LIN {X 0,Y 242.038,Z 353.956,A -85,B 0,C 180,E1 -19224.498,E2 -19224.498} C_VEL
LIN {X 0,Y 241.957,Z 353.973,A -85,B 0,C 180,E1 -19228.478,E2 -19228.478} C_VEL
LIN {X 0,Y 241.972,Z 353.968,A -85,B 0,C 180,E1 -19232.309,E2 -19232.309} C_VEL
LIN {X 0,Y 242.029,Z 353.963,A -85,B 0,C 180,E1 -19236.013,E2 -19236.013} C_VEL
LIN {X 0,Y 242.039,Z 353.959,A -85,B 0,C 180,E1 -19239.608,E2 -19239.608} C_VEL
LIN {X 0,Y 242.166,Z 353.937,A -85,B 0,C 180,E1 -19243.279,E2 -19243.279} C_VEL
LIN {X 0,Y 242.184,Z 353.936,A -85,B 0,C 180,E1 -19248.28,E2 -19248.28} C_VEL
LIN {X 0,Y 242.374,Z 353.905,A -85,B 0,C 180,E1 -19251.664,E2 -19251.664} C_VEL
LIN {X 0,Y 242.4,Z 353.912,A -85,B 0,C 180,E1 -19253.341,E2 -19253.341} C_VEL
LIN {X 0,Y 242.624,Z 353.883,A -85,B 0,C 180,E1 -19258.341,E2 -19258.341} C_VEL
LIN {X 0,Y 242.63,Z 353.872,A -85,B 0,C 180,E1 -19261.66,E2 -19261.66} C_VEL
LIN {X 0,Y 242.401,Z 353.9,A -85,B 0,C 180,E1 -19266.66,E2 -19266.66} C_VEL
LIN {X 0,Y 242.268,Z 353.929,A -85,B 0,C 180,E1 -19270.024,E2 -19270.024} C_VEL
LIN {X 0,Y 242.11,Z 353.946,A -85,B 0,C 180,E1 -19275.145,E2 -19275.145} C_VEL
LIN {X 0,Y 242.019,Z 353.963,A -85,B 0,C 180,E1 -19278.629,E2 -19278.629} C_VEL
LIN {X 0,Y 241.975,Z 353.965,A -85,B 0,C 180,E1 -19282.184,E2 -19282.184} C_VEL
LIN {X 0,Y 241.988,Z 353.96,A -85,B 0,C 180,E1 -19285.827,E2 -19285.827} C_VEL
LIN {X 0,Y 241.965,Z 353.934,A -85,B 0,C 180,E1 -19289.59,E2 -19289.59} C_VEL
LIN {X 0,Y 241.982,Z 353.969,A -85,B 0,C 180,E1 -19293.493,E2 -19293.493} C_VEL
LIN {X 0,Y 241.981,Z 353.944,A -85,B 0,C 180,E1 -19297.584,E2 -19297.584} C_VEL
LIN {X 0,Y 241.974,Z 353.962,A -85,B 0,C 180,E1 -19298.682,E2 -19298.682} C_VEL
LIN {X 0,Y 242.898,Z 356.753,A -85,B 0,C 180,E1 -19299.067,E2 -19299.067} C_VEL
LIN {X 0,Y 245.049,Z 359.01,A -85,B 0,C 180,E1 -19299.727,E2 -19299.727} C_VEL
LIN {X 0,Y 247.606,Z 362.894,A -85,B 0,C 180,E1 -19300.538,E2 -19300.538} C_VEL
LIN {X 0,Y 248.987,Z 364.649,A -85,B 0,C 180,E1 -19300.949,E2 -19300.949} C_VEL
LIN {X 0,Y 256.882,Z 376.241,A -85,B 0,C 180,E1 -19303.223,E2 -19303.223} C_VEL
LIN {X 0,Y 264.702,Z 390.021,A -85,B 0,C 180,E1 -19305.346,E2 -19305.346} C_VEL
LIN {X 0,Y 272.156,Z 405.107,A -85,B 0,C 180,E1 -19307.261,E2 -19307.261} C_VEL
LIN {X 0,Y 274.978,Z 411.557,A -85,B 0,C 180,E1 -19307.97,E2 -19307.97} C_VEL
LIN {X 0,Y 271.334,Z 488.503,A -85,B 0,C 180,E1 -19309.947,E2 -19309.947} C_VEL
LIN {X 0,Y 270.043,Z 502.422,A -85,B 0,C 180,E1 -19310.566,E2 -19310.566} C_VEL
LIN {X 0,Y 267.985,Z 516.616,A -85,B 0,C 180,E1 -19311.475,E2 -19311.475} C_VEL
LIN {X 0,Y 265.359,Z 530.29,A -85,B 0,C 180,E1 -19312.664,E2 -19312.664} C_VEL
LIN {X 0,Y 262.577,Z 543.151,A -85,B 0,C 180,E1 -19314.162,E2 -19314.162} C_VEL
LIN {X 0,Y 259.471,Z 554.546,A -85,B 0,C 180,E1 -19315.803,E2 -19315.803} C_VEL
LIN {X 0,Y 256.414,Z 565.005,A -85,B 0,C 180,E1 -19317.692,E2 -19317.692} C_VEL
LIN {X 0,Y 253.24,Z 575.381,A -85,B 0,C 180,E1 -19320.03,E2 -19320.03} C_VEL
LIN {X 0,Y 250.217,Z 583.915,A -85,B 0,C 180,E1 -19322.39,E2 -19322.39} C_VEL
LIN {X 0,Y 247.608,Z 590.992,A -85,B 0,C 180,E1 -19324.801,E2 -19324.801} C_VEL
LIN {X 0,Y 245.473,Z 596.839,A -85,B 0,C 180,E1 -19327.262,E2 -19327.262} C_VEL
LIN {X 0,Y 243.185,Z 603.065,A -85,B 0,C 180,E1 -19330.588,E2 -19330.588} C_VEL
LIN {X 0,Y 241.694,Z 607.276,A -85,B 0,C 180,E1 -19333.656,E2 -19333.656} C_VEL
LIN {X 0,Y 240.668,Z 610.028,A -85,B 0,C 180,E1 -19336.49,E2 -19336.49} C_VEL
LIN {X 0,Y 239.974,Z 612.057,A -85,B 0,C 180,E1 -19339.879,E2 -19339.879} C_VEL
LIN {X 0,Y 239.855,Z 612.741,A -85,B 0,C 180,E1 -19343.269,E2 -19343.269} C_VEL
LIN {X 0,Y 239.803,Z 612.535,A -85,B 0,C 180,E1 -19345.18,E2 -19345.18} C_VEL
LIN {X 0,Y 239.895,Z 611.292,A -85,B 0,C 180,E1 -19348.321,E2 -19348.321} C_VEL
LIN {X 0,Y 240.147,Z 608.654,A -85,B 0,C 180,E1 -19351.677,E2 -19351.677} C_VEL
LIN {X 0,Y 240.892,Z 604.604,A -85,B 0,C 180,E1 -19355.021,E2 -19355.021} C_VEL
LIN {X 0,Y 242.269,Z 599.01,A -85,B 0,C 180,E1 -19358.34,E2 -19358.34} C_VEL
LIN {X 0,Y 243.69,Z 593.257,A -85,B 0,C 180,E1 -19360.994,E2 -19360.994} C_VEL
LIN {X 0,Y 245.286,Z 586.113,A -85,B 0,C 180,E1 -19363.673,E2 -19363.673} C_VEL
LIN {X 0,Y 247.415,Z 578.179,A -85,B 0,C 180,E1 -19366.079,E2 -19366.079} C_VEL
LIN {X 0,Y 249.976,Z 568.609,A -85,B 0,C 180,E1 -19368.439,E2 -19368.439} C_VEL
LIN {X 0,Y 252.356,Z 558.026,A -85,B 0,C 180,E1 -19370.585,E2 -19370.585} C_VEL
LIN {X 0,Y 254.879,Z 546.305,A -85,B 0,C 180,E1 -19372.494,E2 -19372.494} C_VEL
LIN {X 0,Y 257.449,Z 533.24,A -85,B 0,C 180,E1 -19374.172,E2 -19374.172} C_VEL
LIN {X 0,Y 259.472,Z 520.349,A -85,B 0,C 180,E1 -19375.467,E2 -19375.467} C_VEL
LIN {X 0,Y 261.277,Z 506.3,A -85,B 0,C 180,E1 -19376.51,E2 -19376.51} C_VEL
LIN {X 0,Y 262.486,Z 491.876,A -85,B 0,C 180,E1 -19377.266,E2 -19377.266} C_VEL
LIN {X 0,Y 263.407,Z 473.595,A -85,B 0,C 180,E1 -19377.827,E2 -19377.827} C_VEL
LIN {X 0,Y 266.21,Z 403.022,A -85,B 0,C 180,E1 -19379.659,E2 -19379.659} C_VEL
LIN {X 0,Y 259.511,Z 386.758,A -85,B 0,C 180,E1 -19381.142,E2 -19381.142} C_VEL
LIN {X 0,Y 253.103,Z 373.357,A -85,B 0,C 180,E1 -19382.587,E2 -19382.587} C_VEL
LIN {X 0,Y 246.089,Z 361.534,A -85,B 0,C 180,E1 -19384.184,E2 -19384.184} C_VEL
LIN {X 0,Y 243.888,Z 357.969,A -85,B 0,C 180,E1 -19384.706,E2 -19384.706} C_VEL
LIN {X 0,Y 242.341,Z 355.359,A -85,B 0,C 180,E1 -19385.085,E2 -19385.085} C_VEL
LIN {X 0,Y 242.002,Z 353.964,A -85,B 0,C 180,E1 -19385.222,E2 -19385.222} C_VEL
LIN {X 0,Y 241.996,Z 353.966,A -85,B 0,C 180,E1 -19388.359,E2 -19388.359} C_VEL
LIN {X 0,Y 241.903,Z 353.978,A -85,B 0,C 180,E1 -19393.42,E2 -19393.42} C_VEL
LIN {X 0,Y 241.909,Z 353.971,A -85,B 0,C 180,E1 -19398.071,E2 -19398.071} C_VEL
LIN {X 0,Y 241.968,Z 353.961,A -85,B 0,C 180,E1 -19402.413,E2 -19402.413} C_VEL
LIN {X 0,Y 241.981,Z 353.958,A -85,B 0,C 180,E1 -19406.507,E2 -19406.507} C_VEL
LIN {X 0,Y 241.973,Z 353.966,A -85,B 0,C 180,E1 -19410.615,E2 -19410.615} C_VEL
LIN {X 0,Y 241.998,Z 353.961,A -85,B 0,C 180,E1 -19414.197,E2 -19414.197} C_VEL
LIN {X 0,Y 241.989,Z 353.939,A -85,B 0,C 180,E1 -19418.337,E2 -19418.337} C_VEL
LIN {X 0,Y 242.108,Z 353.95,A -85,B 0,C 180,E1 -19423.324,E2 -19423.324} C_VEL
LIN {X 0,Y 242.159,Z 353.906,A -85,B 0,C 180,E1 -19428.278,E2 -19428.278} C_VEL
LIN {X 0,Y 242.384,Z 353.905,A -85,B 0,C 180,E1 -19431.664,E2 -19431.664} C_VEL
LIN {X 0,Y 242.235,Z 353.933,A -85,B 0,C 180,E1 -19435.006,E2 -19435.006} C_VEL
LIN {X 0,Y 242.63,Z 353.889,A -85,B 0,C 180,E1 -19438.34,E2 -19438.34} C_VEL
LIN {X 0,Y 242.606,Z 353.88,A -85,B 0,C 180,E1 -19441.115,E2 -19441.115} C_VEL
LIN {X 0,Y 242.289,Z 353.924,A -85,B 0,C 180,E1 -19442.04,E2 -19442.04} C_VEL
LIN {X 0,Y 240.898,Z 354.103,A -85,B 0,C 180,E1 -19443.403,E2 -19443.403} C_VEL
LIN {X 0,Y 236.439,Z 354.654,A -85,B 0,C 180,E1 -19446.579,E2 -19446.579} C_VEL
LIN {X 0,Y 235.387,Z 354.791,A -85,B 0,C 180,E1 -19448.006,E2 -19448.006} C_VEL
LIN {X 0,Y 235.317,Z 354.795,A -85,B 0,C 180,E1 -19448.49,E2 -19448.49} C_VEL
LIN {X 0,Y 235.116,Z 354.825,A -85,B 0,C 180,E1 -19452.077,E2 -19452.077} C_VEL
LIN {X 0,Y 235.098,Z 354.824,A -85,B 0,C 180,E1 -19456.94,E2 -19456.94} C_VEL
LIN {X 0,Y 234.979,Z 354.835,A -85,B 0,C 180,E1 -19462,E2 -19462} C_VEL
LIN {X 0,Y 234.964,Z 354.842,A -85,B 0,C 180,E1 -19466.658,E2 -19466.658} C_VEL
LIN {X 0,Y 234.904,Z 354.853,A -85,B 0,C 180,E1 -19470.571,E2 -19470.571} C_VEL
LIN {X 0,Y 234.961,Z 354.846,A -85,B 0,C 180,E1 -19474.632,E2 -19474.632} C_VEL
LIN {X 0,Y 234.942,Z 354.844,A -85,B 0,C 180,E1 -19478.944,E2 -19478.944} C_VEL
LIN {X 0,Y 234.888,Z 354.854,A -85,B 0,C 180,E1 -19483.485,E2 -19483.485} C_VEL
LIN {X 0,Y 234.902,Z 355.016,A -85,B 0,C 180,E1 -19485.525,E2 -19485.525} C_VEL
LIN {X 0,Y 237.054,Z 362.356,A -85,B 0,C 180,E1 -19488.815,E2 -19488.815} C_VEL
LIN {X 0,Y 244.613,Z 376.813,A -85,B 0,C 180,E1 -19490.744,E2 -19490.744} C_VEL
LIN {X 0,Y 251.022,Z 390.294,A -85,B 0,C 180,E1 -19492.296,E2 -19492.296} C_VEL
LIN {X 0,Y 257.884,Z 407.058,A -85,B 0,C 180,E1 -19493.92,E2 -19493.92} C_VEL
LIN {X 0,Y 259.65,Z 421.423,A -85,B 0,C 180,E1 -19494.645,E2 -19494.645} C_VEL
LIN {X 0,Y 256.29,Z 501.166,A -85,B 0,C 180,E1 -19496.798,E2 -19496.798} C_VEL
LIN {X 0,Y 254.887,Z 515.707,A -85,B 0,C 180,E1 -19497.474,E2 -19497.474} C_VEL
LIN {X 0,Y 253.16,Z 529.091,A -85,B 0,C 180,E1 -19498.399,E2 -19498.399} C_VEL
LIN {X 0,Y 250.732,Z 543.076,A -85,B 0,C 180,E1 -19499.699,E2 -19499.699} C_VEL
LIN {X 0,Y 248.266,Z 555.601,A -85,B 0,C 180,E1 -19501.233,E2 -19501.233} C_VEL
LIN {X 0,Y 245.687,Z 567.041,A -85,B 0,C 180,E1 -19502.992,E2 -19502.992} C_VEL
LIN {X 0,Y 242.827,Z 578.526,A -85,B 0,C 180,E1 -19505.186,E2 -19505.186} C_VEL
LIN {X 0,Y 240.13,Z 588.763,A -85,B 0,C 180,E1 -19507.637,E2 -19507.637} C_VEL
LIN {X 0,Y 237.867,Z 597.252,A -85,B 0,C 180,E1 -19510.137,E2 -19510.137} C_VEL
LIN {X 0,Y 236.284,Z 604.343,A -85,B 0,C 180,E1 -19512.696,E2 -19512.696} C_VEL
LIN {X 0,Y 234.84,Z 610.185,A -85,B 0,C 180,E1 -19515.263,E2 -19515.263} C_VEL
LIN {X 0,Y 233.749,Z 614.988,A -85,B 0,C 180,E1 -19517.85,E2 -19517.85} C_VEL
LIN {X 0,Y 233.056,Z 619.962,A -85,B 0,C 180,E1 -19521.328,E2 -19521.328} C_VEL
LIN {X 0,Y 232.742,Z 623.417,A -85,B 0,C 180,E1 -19524.803,E2 -19524.803} C_VEL
LIN {X 0,Y 232.753,Z 625.46,A -85,B 0,C 180,E1 -19528.27,E2 -19528.27} C_VEL
LIN {X 0,Y 232.822,Z 625.969,A -85,B 0,C 180,E1 -19530,E2 -19530} C_VEL
LIN {X 0,Y 232.666,Z 625.964,A -85,B 0,C 180,E1 -19533.464,E2 -19533.464} C_VEL
LIN {X 0,Y 232.813,Z 624.622,A -85,B 0,C 180,E1 -19536.935,E2 -19536.935} C_VEL
LIN {X 0,Y 233.441,Z 621.922,A -85,B 0,C 180,E1 -19540.407,E2 -19540.407} C_VEL
LIN {X 0,Y 234.628,Z 617.798,A -85,B 0,C 180,E1 -19543.865,E2 -19543.865} C_VEL
LIN {X 0,Y 236.072,Z 613.734,A -85,B 0,C 180,E1 -19546.429,E2 -19546.429} C_VEL
LIN {X 0,Y 237.755,Z 608.673,A -85,B 0,C 180,E1 -19548.975,E2 -19548.975} C_VEL
LIN {X 0,Y 240.452,Z 601.469,A -85,B 0,C 180,E1 -19551.88,E2 -19551.88} C_VEL
LIN {X 0,Y 243.252,Z 593.941,A -85,B 0,C 180,E1 -19554.312,E2 -19554.312} C_VEL
LIN {X 0,Y 246.49,Z 584.922,A -85,B 0,C 180,E1 -19556.684,E2 -19556.684} C_VEL
LIN {X 0,Y 250.201,Z 574.018,A -85,B 0,C 180,E1 -19558.983,E2 -19558.983} C_VEL
LIN {X 0,Y 253.683,Z 562.104,A -85,B 0,C 180,E1 -19560.994,E2 -19560.994} C_VEL
LIN {X 0,Y 256.677,Z 550.815,A -85,B 0,C 180,E1 -19562.503,E2 -19562.503} C_VEL
LIN {X 0,Y 259.41,Z 539.143,A -85,B 0,C 180,E1 -19563.738,E2 -19563.738} C_VEL
LIN {X 0,Y 261.892,Z 526.517,A -85,B 0,C 180,E1 -19564.768,E2 -19564.768} C_VEL
LIN {X 0,Y 263.979,Z 512.328,A -85,B 0,C 180,E1 -19565.619,E2 -19565.619} C_VEL
LIN {X 0,Y 265.367,Z 498.18,A -85,B 0,C 180,E1 -19566.181,E2 -19566.181} C_VEL
LIN {X 0,Y 268.956,Z 424.085,A -85,B 0,C 180,E1 -19568.102,E2 -19568.102} C_VEL
LIN {X 0,Y 268.104,Z 419.277,A -85,B 0,C 180,E1 -19568.421,E2 -19568.421} C_VEL
LIN {X 0,Y 260.963,Z 403.057,A -85,B 0,C 180,E1 -19570.361,E2 -19570.361} C_VEL
LIN {X 0,Y 253.943,Z 389.349,A -85,B 0,C 180,E1 -19572.354,E2 -19572.354} C_VEL
LIN {X 0,Y 248.816,Z 380.347,A -85,B 0,C 180,E1 -19573.887,E2 -19573.887} C_VEL
LIN {X 0,Y 243.257,Z 371.277,A -85,B 0,C 180,E1 -19575.647,E2 -19575.647} C_VEL
LIN {X 0,Y 239.877,Z 366.033,A -85,B 0,C 180,E1 -19576.777,E2 -19576.777} C_VEL
LIN {X 0,Y 237.106,Z 361.609,A -85,B 0,C 180,E1 -19577.752,E2 -19577.752} C_VEL
LIN {X 0,Y 234.966,Z 354.837,A -85,B 0,C 180,E1 -19581.637,E2 -19581.637} C_VEL
LIN {X 0,Y 234.961,Z 354.843,A -85,B 0,C 180,E1 -19585.368,E2 -19585.368} C_VEL
LIN {X 0,Y 234.901,Z 354.844,A -85,B 0,C 180,E1 -19589.428,E2 -19589.428} C_VEL
LIN {X 0,Y 234.97,Z 354.831,A -85,B 0,C 180,E1 -19593.807,E2 -19593.807} C_VEL
LIN {X 0,Y 235,Z 354.831,A -85,B 0,C 180,E1 -19598.969,E2 -19598.969} C_VEL
LIN {X 0,Y 235.099,Z 354.815,A -85,B 0,C 180,E1 -19603.06,E2 -19603.06} C_VEL
LIN {X 0,Y 235.117,Z 354.813,A -85,B 0,C 180,E1 -19607.923,E2 -19607.923} C_VEL
LIN {X 0,Y 235.314,Z 354.784,A -85,B 0,C 180,E1 -19611.412,E2 -19611.412} C_VEL
LIN {X 0,Y 235.351,Z 354.788,A -85,B 0,C 180,E1 -19613.14,E2 -19613.14} C_VEL
LIN {X 0,Y 235.582,Z 354.759,A -85,B 0,C 180,E1 -19618.291,E2 -19618.291} C_VEL
LIN {X 0,Y 235.59,Z 354.749,A -85,B 0,C 180,E1 -19621.71,E2 -19621.71} C_VEL
LIN {X 0,Y 235.352,Z 354.777,A -85,B 0,C 180,E1 -19626.861,E2 -19626.861} C_VEL
LIN {X 0,Y 235.213,Z 354.806,A -85,B 0,C 180,E1 -19630.328,E2 -19630.328} C_VEL
LIN {X 0,Y 235.046,Z 354.821,A -85,B 0,C 180,E1 -19635.612,E2 -19635.612} C_VEL
LIN {X 0,Y 234.961,Z 354.84,A -85,B 0,C 180,E1 -19639.21,E2 -19639.21} C_VEL
LIN {X 0,Y 234.91,Z 354.849,A -85,B 0,C 180,E1 -19642.889,E2 -19642.889} C_VEL
LIN {X 0,Y 234.924,Z 354.847,A -85,B 0,C 180,E1 -19646.664,E2 -19646.664} C_VEL
LIN {X 0,Y 234.897,Z 354.811,A -85,B 0,C 180,E1 -19650.573,E2 -19650.573} C_VEL
LIN {X 0,Y 234.927,Z 354.833,A -85,B 0,C 180,E1 -19654.639,E2 -19654.639} C_VEL
LIN {X 0,Y 234.908,Z 354.82,A -85,B 0,C 180,E1 -19656.705,E2 -19656.705} C_VEL
LIN {X 0,Y 235.939,Z 357.712,A -85,B 0,C 180,E1 -19657.167,E2 -19657.167} C_VEL
LIN {X 0,Y 238.538,Z 360.489,A -85,B 0,C 180,E1 -19658.041,E2 -19658.041} C_VEL
LIN {X 0,Y 240.472,Z 363.618,A -85,B 0,C 180,E1 -19658.716,E2 -19658.716} C_VEL
LIN {X 0,Y 242.068,Z 365.467,A -85,B 0,C 180,E1 -19659.227,E2 -19659.227} C_VEL
LIN {X 0,Y 244.768,Z 369.133,A -85,B 0,C 180,E1 -19660.087,E2 -19660.087} C_VEL
LIN {X 0,Y 252.844,Z 381.166,A -85,B 0,C 180,E1 -19662.518,E2 -19662.518} C_VEL
LIN {X 0,Y 260.839,Z 395.564,A -85,B 0,C 180,E1 -19664.778,E2 -19664.778} C_VEL
LIN {X 0,Y 268.043,Z 410.591,A -85,B 0,C 180,E1 -19666.705,E2 -19666.705} C_VEL
LIN {X 0,Y 269.406,Z 413.651,A -85,B 0,C 180,E1 -19667.06,E2 -19667.06} C_VEL
LIN {X 0,Y 265.701,Z 489.22,A -85,B 0,C 180,E1 -19669.043,E2 -19669.043} C_VEL
LIN {X 0,Y 264.357,Z 502.967,A -85,B 0,C 180,E1 -19669.67,E2 -19669.67} C_VEL
LIN {X 0,Y 262.227,Z 517.071,A -85,B 0,C 180,E1 -19670.591,E2 -19670.591} C_VEL
LIN {X 0,Y 259.681,Z 529.841,A -85,B 0,C 180,E1 -19671.708,E2 -19671.708} C_VEL
LIN {X 0,Y 256.799,Z 542.794,A -85,B 0,C 180,E1 -19673.225,E2 -19673.225} C_VEL
LIN {X 0,Y 253.572,Z 554.288,A -85,B 0,C 180,E1 -19674.893,E2 -19674.893} C_VEL
LIN {X 0,Y 250.36,Z 564.825,A -85,B 0,C 180,E1 -19676.811,E2 -19676.811} C_VEL
LIN {X 0,Y 247.031,Z 575.275,A -85,B 0,C 180,E1 -19679.196,E2 -19679.196} C_VEL
LIN {X 0,Y 243.834,Z 583.862,A -85,B 0,C 180,E1 -19681.603,E2 -19681.603} C_VEL
LIN {X 0,Y 241.105,Z 590.976,A -85,B 0,C 180,E1 -19684.072,E2 -19684.072} C_VEL
LIN {X 0,Y 238.826,Z 596.864,A -85,B 0,C 180,E1 -19686.592,E2 -19686.592} C_VEL
LIN {X 0,Y 236.398,Z 603.13,A -85,B 0,C 180,E1 -19690.008,E2 -19690.008} C_VEL
LIN {X 0,Y 234.69,Z 607.639,A -85,B 0,C 180,E1 -19693.392,E2 -19693.392} C_VEL
LIN {X 0,Y 233.703,Z 610.159,A -85,B 0,C 180,E1 -19696.079,E2 -19696.079} C_VEL
LIN {X 0,Y 232.923,Z 612.221,A -85,B 0,C 180,E1 -19699.57,E2 -19699.57} C_VEL
LIN {X 0,Y 232.764,Z 612.936,A -85,B 0,C 180,E1 -19703.063,E2 -19703.063} C_VEL
LIN {X 0,Y 232.712,Z 612.339,A -85,B 0,C 180,E1 -19706.537,E2 -19706.537} C_VEL
LIN {X 0,Y 232.91,Z 610.414,A -85,B 0,C 180,E1 -19710,E2 -19710} C_VEL
LIN {X 0,Y 233.377,Z 607.118,A -85,B 0,C 180,E1 -19713.453,E2 -19713.453} C_VEL
LIN {X 0,Y 234.495,Z 602.349,A -85,B 0,C 180,E1 -19716.885,E2 -19716.885} C_VEL
LIN {X 0,Y 236.13,Z 595.966,A -85,B 0,C 180,E1 -19720.287,E2 -19720.287} C_VEL
LIN {X 0,Y 237.891,Z 588.874,A -85,B 0,C 180,E1 -19723.236,E2 -19723.236} C_VEL
LIN {X 0,Y 239.798,Z 581.454,A -85,B 0,C 180,E1 -19725.73,E2 -19725.73} C_VEL
LIN {X 0,Y 242.391,Z 572.522,A -85,B 0,C 180,E1 -19728.161,E2 -19728.161} C_VEL
LIN {X 0,Y 245.136,Z 561.728,A -85,B 0,C 180,E1 -19730.561,E2 -19730.561} C_VEL
LIN {X 0,Y 247.352,Z 551.946,A -85,B 0,C 180,E1 -19732.335,E2 -19732.335} C_VEL
LIN {X 0,Y 249.852,Z 540.177,A -85,B 0,C 180,E1 -19734.071,E2 -19734.071} C_VEL
LIN {X 0,Y 252.17,Z 527.194,A -85,B 0,C 180,E1 -19735.594,E2 -19735.594} C_VEL
LIN {X 0,Y 254.239,Z 513.502,A -85,B 0,C 180,E1 -19736.804,E2 -19736.804} C_VEL
LIN {X 0,Y 255.866,Z 498.988,A -85,B 0,C 180,E1 -19737.725,E2 -19737.725} C_VEL
LIN {X 0,Y 256.858,Z 484.876,A -85,B 0,C 180,E1 -19738.319,E2 -19738.319} C_VEL
LIN {X 0,Y 260.207,Z 404.979,A -85,B 0,C 180,E1 -19740.445,E2 -19740.445} C_VEL
LIN {X 0,Y 253.509,Z 388.698,A -85,B 0,C 180,E1 -19742,E2 -19742} C_VEL
LIN {X 0,Y 247.691,Z 376.596,A -85,B 0,C 180,E1 -19743.371,E2 -19743.371} C_VEL
LIN {X 0,Y 239.335,Z 362.699,A -85,B 0,C 180,E1 -19745.374,E2 -19745.374} C_VEL
LIN {X 0,Y 236.857,Z 358.906,A -85,B 0,C 180,E1 -19745.993,E2 -19745.993} C_VEL
LIN {X 0,Y 235.378,Z 356.62,A -85,B 0,C 180,E1 -19746.373,E2 -19746.373} C_VEL
LIN {X 0,Y 234.908,Z 354.846,A -85,B 0,C 180,E1 -19746.559,E2 -19746.559} C_VEL
LIN {X 0,Y 234.914,Z 354.845,A -85,B 0,C 180,E1 -19748.935,E2 -19748.935} C_VEL
LIN {X 0,Y 234.856,Z 354.856,A -85,B 0,C 180,E1 -19753.494,E2 -19753.494} C_VEL
LIN {X 0,Y 234.856,Z 354.855,A -85,B 0,C 180,E1 -19756.506,E2 -19756.506} C_VEL
LIN {X 0,Y 234.92,Z 354.846,A -85,B 0,C 180,E1 -19761.078,E2 -19761.078} C_VEL
LIN {X 0,Y 234.924,Z 354.846,A -85,B 0,C 180,E1 -19765.36,E2 -19765.36} C_VEL
LIN {X 0,Y 234.897,Z 354.85,A -85,B 0,C 180,E1 -19769.427,E2 -19769.427} C_VEL
LIN {X 0,Y 234.942,Z 354.837,A -85,B 0,C 180,E1 -19773.821,E2 -19773.821} C_VEL
LIN {X 0,Y 234.939,Z 354.81,A -85,B 0,C 180,E1 -19778.962,E2 -19778.962} C_VEL
LIN {X 0,Y 235.052,Z 354.828,A -85,B 0,C 180,E1 -19783.097,E2 -19783.097} C_VEL
LIN {X 0,Y 235.091,Z 354.788,A -85,B 0,C 180,E1 -19787.92,E2 -19787.92} C_VEL
LIN {X 0,Y 235.317,Z 354.778,A -85,B 0,C 180,E1 -19791.411,E2 -19791.411} C_VEL
LIN {X 0,Y 235.356,Z 354.792,A -85,B 0,C 180,E1 -19793.139,E2 -19793.139} C_VEL
LIN {X 0,Y 235.589,Z 354.765,A -85,B 0,C 180,E1 -19798.29,E2 -19798.29} C_VEL
LIN {X 0,Y 235.582,Z 354.756,A -85,B 0,C 180,E1 -19801.709,E2 -19801.709} C_VEL
LIN {X 0,Y 235.356,Z 354.791,A -85,B 0,C 180,E1 -19806.86,E2 -19806.86} C_VEL
LIN {X 0,Y 235.317,Z 354.795,A -85,B 0,C 180,E1 -19808.49,E2 -19808.49} C_VEL
LIN {X 0,Y 234.681,Z 354.883,A -85,B 0,C 180,E1 -19809.915,E2 -19809.915} C_VEL
LIN {X 0,Y 231.793,Z 355.251,A -85,B 0,C 180,E1 -19812.238,E2 -19812.238} C_VEL
LIN {X 0,Y 229.286,Z 355.561,A -85,B 0,C 180,E1 -19814.133,E2 -19814.133} C_VEL
LIN {X 0,Y 228.17,Z 355.693,A -85,B 0,C 180,E1 -19815.605,E2 -19815.605} C_VEL
LIN {X 0,Y 228.06,Z 355.703,A -85,B 0,C 180,E1 -19816.105,E2 -19816.105} C_VEL
LIN {X 0,Y 227.94,Z 355.717,A -85,B 0,C 180,E1 -19819.825,E2 -19819.825} C_VEL
LIN {X 0,Y 227.907,Z 355.721,A -85,B 0,C 180,E1 -19823.633,E2 -19823.633} C_VEL
LIN {X 0,Y 227.869,Z 355.729,A -85,B 0,C 180,E1 -19827.557,E2 -19827.557} C_VEL
LIN {X 0,Y 227.861,Z 355.728,A -85,B 0,C 180,E1 -19831.623,E2 -19831.623} C_VEL
LIN {X 0,Y 227.901,Z 355.722,A -85,B 0,C 180,E1 -19835.868,E2 -19835.868} C_VEL
LIN {X 0,Y 227.834,Z 355.733,A -85,B 0,C 180,E1 -19840.375,E2 -19840.375} C_VEL
LIN {X 0,Y 227.865,Z 355.854,A -85,B 0,C 180,E1 -19844.376,E2 -19844.376} C_VEL
LIN {X 0,Y 229.575,Z 361.881,A -85,B 0,C 180,E1 -19847.283,E2 -19847.283} C_VEL
LIN {X 0,Y 232.072,Z 366.339,A -85,B 0,C 180,E1 -19847.978,E2 -19847.978} C_VEL
LIN {X 0,Y 239.259,Z 379.873,A -85,B 0,C 180,E1 -19849.891,E2 -19849.891} C_VEL
LIN {X 0,Y 245.885,Z 394.148,A -85,B 0,C 180,E1 -19851.581,E2 -19851.581} C_VEL
LIN {X 0,Y 252.218,Z 409.727,A -85,B 0,C 180,E1 -19853.148,E2 -19853.148} C_VEL
LIN {X 0,Y 253.714,Z 421.922,A -85,B 0,C 180,E1 -19853.788,E2 -19853.788} C_VEL
LIN {X 0,Y 250.258,Z 500.69,A -85,B 0,C 180,E1 -19855.951,E2 -19855.951} C_VEL
LIN {X 0,Y 248.816,Z 515.323,A -85,B 0,C 180,E1 -19856.639,E2 -19856.639} C_VEL
LIN {X 0,Y 247.122,Z 528.187,A -85,B 0,C 180,E1 -19857.534,E2 -19857.534} C_VEL
LIN {X 0,Y 244.962,Z 540.549,A -85,B 0,C 180,E1 -19858.667,E2 -19858.667} C_VEL
LIN {X 0,Y 242.29,Z 553.511,A -85,B 0,C 180,E1 -19860.215,E2 -19860.215} C_VEL
LIN {X 0,Y 239.655,Z 565.291,A -85,B 0,C 180,E1 -19862.017,E2 -19862.017} C_VEL
LIN {X 0,Y 236.856,Z 576.056,A -85,B 0,C 180,E1 -19864.045,E2 -19864.045} C_VEL
LIN {X 0,Y 233.962,Z 586.723,A -85,B 0,C 180,E1 -19866.546,E2 -19866.546} C_VEL
LIN {X 0,Y 231.535,Z 595.524,A -85,B 0,C 180,E1 -19869.105,E2 -19869.105} C_VEL
LIN {X 0,Y 229.734,Z 602.295,A -85,B 0,C 180,E1 -19871.503,E2 -19871.503} C_VEL
LIN {X 0,Y 228.365,Z 608.011,A -85,B 0,C 180,E1 -19873.92,E2 -19873.92} C_VEL
LIN {X 0,Y 227.122,Z 613.196,A -85,B 0,C 180,E1 -19876.581,E2 -19876.581} C_VEL
LIN {X 0,Y 226.127,Z 618.599,A -85,B 0,C 180,E1 -19880.158,E2 -19880.158} C_VEL
LIN {X 0,Y 225.758,Z 621.6,A -85,B 0,C 180,E1 -19882.847,E2 -19882.847} C_VEL
LIN {X 0,Y 225.61,Z 624.365,A -85,B 0,C 180,E1 -19886.428,E2 -19886.428} C_VEL
LIN {X 0,Y 225.734,Z 625.75,A -85,B 0,C 180,E1 -19890,E2 -19890} C_VEL
LIN {X 0,Y 225.656,Z 625.93,A -85,B 0,C 180,E1 -19891.785,E2 -19891.785} C_VEL
LIN {X 0,Y 225.641,Z 625.284,A -85,B 0,C 180,E1 -19895.362,E2 -19895.362} C_VEL
LIN {X 0,Y 226.017,Z 623.298,A -85,B 0,C 180,E1 -19898.944,E2 -19898.944} C_VEL
LIN {X 0,Y 226.912,Z 619.923,A -85,B 0,C 180,E1 -19902.522,E2 -19902.522} C_VEL
LIN {X 0,Y 228.714,Z 615.076,A -85,B 0,C 180,E1 -19906.055,E2 -19906.055} C_VEL
LIN {X 0,Y 231.029,Z 608.611,A -85,B 0,C 180,E1 -19909.55,E2 -19909.55} C_VEL
LIN {X 0,Y 233.852,Z 601.439,A -85,B 0,C 180,E1 -19912.531,E2 -19912.531} C_VEL
LIN {X 0,Y 236.795,Z 593.948,A -85,B 0,C 180,E1 -19915.02,E2 -19915.02} C_VEL
LIN {X 0,Y 240.168,Z 584.971,A -85,B 0,C 180,E1 -19917.445,E2 -19917.445} C_VEL
LIN {X 0,Y 243.993,Z 574.184,A -85,B 0,C 180,E1 -19919.777,E2 -19919.777} C_VEL
LIN {X 0,Y 247.631,Z 562.293,A -85,B 0,C 180,E1 -19921.839,E2 -19921.839} C_VEL
LIN {X 0,Y 251.091,Z 549.529,A -85,B 0,C 180,E1 -19923.56,E2 -19923.56} C_VEL
LIN {X 0,Y 253.943,Z 537.602,A -85,B 0,C 180,E1 -19924.807,E2 -19924.807} C_VEL
LIN {X 0,Y 256.513,Z 524.56,A -85,B 0,C 180,E1 -19925.848,E2 -19925.848} C_VEL
LIN {X 0,Y 258.609,Z 510.522,A -85,B 0,C 180,E1 -19926.658,E2 -19926.658} C_VEL
LIN {X 0,Y 259.932,Z 496.145,A -85,B 0,C 180,E1 -19927.213,E2 -19927.213} C_VEL
LIN {X 0,Y 263.496,Z 425.204,A -85,B 0,C 180,E1 -19929.07,E2 -19929.07} C_VEL
LIN {X 0,Y 262.854,Z 422.033,A -85,B 0,C 180,E1 -19929.305,E2 -19929.305} C_VEL
LIN {X 0,Y 255.794,Z 405.94,A -85,B 0,C 180,E1 -19931.318,E2 -19931.318} C_VEL
LIN {X 0,Y 248.201,Z 391.042,A -85,B 0,C 180,E1 -19933.599,E2 -19933.599} C_VEL
LIN {X 0,Y 240.086,Z 377.145,A -85,B 0,C 180,E1 -19936.227,E2 -19936.227} C_VEL
LIN {X 0,Y 235.793,Z 370.644,A -85,B 0,C 180,E1 -19937.712,E2 -19937.712} C_VEL
LIN {X 0,Y 232.797,Z 366.015,A -85,B 0,C 180,E1 -19938.815,E2 -19938.815} C_VEL
LIN {X 0,Y 229.889,Z 361.676,A -85,B 0,C 180,E1 -19939.931,E2 -19939.931} C_VEL
LIN {X 0,Y 229.535,Z 360.839,A -85,B 0,C 180,E1 -19940.158,E2 -19940.158} C_VEL
LIN {X 0,Y 227.926,Z 355.711,A -85,B 0,C 180,E1 -19943.455,E2 -19943.455} C_VEL
LIN {X 0,Y 227.89,Z 355.716,A -85,B 0,C 180,E1 -19946.374,E2 -19946.374} C_VEL
LIN {X 0,Y 227.879,Z 355.716,A -85,B 0,C 180,E1 -19950.432,E2 -19950.432} C_VEL
LIN {X 0,Y 227.904,Z 355.712,A -85,B 0,C 180,E1 -19954.423,E2 -19954.423} C_VEL
LIN {X 0,Y 227.957,Z 355.703,A -85,B 0,C 180,E1 -19958.287,E2 -19958.287} C_VEL
LIN {X 0,Y 228.037,Z 355.693,A -85,B 0,C 180,E1 -19962.826,E2 -19962.826} C_VEL
LIN {X 0,Y 228.075,Z 355.687,A -85,B 0,C 180,E1 -19967.544,E2 -19967.544} C_VEL
LIN {X 0,Y 228.255,Z 355.664,A -85,B 0,C 180,E1 -19971.145,E2 -19971.145} C_VEL
LIN {X 0,Y 228.304,Z 355.663,A -85,B 0,C 180,E1 -19972.927,E2 -19972.927} C_VEL
LIN {X 0,Y 228.54,Z 355.635,A -85,B 0,C 180,E1 -19978.238,E2 -19978.238} C_VEL
LIN {X 0,Y 228.548,Z 355.625,A -85,B 0,C 180,E1 -19981.763,E2 -19981.763} C_VEL
LIN {X 0,Y 228.305,Z 355.655,A -85,B 0,C 180,E1 -19987.074,E2 -19987.074} C_VEL
LIN {X 0,Y 228.143,Z 355.682,A -85,B 0,C 180,E1 -19990.652,E2 -19990.652} C_VEL
LIN {X 0,Y 228.003,Z 355.696,A -85,B 0,C 180,E1 -19996.107,E2 -19996.107} C_VEL
LIN {X 0,Y 227.921,Z 355.71,A -85,B 0,C 180,E1 -20001.718,E2 -20001.718} C_VEL
LIN {X 0,Y 227.903,Z 355.722,A -85,B 0,C 180,E1 -20006.581,E2 -20006.581} C_VEL
LIN {X 0,Y 227.872,Z 355.685,A -85,B 0,C 180,E1 -20010.279,E2 -20010.279} C_VEL
LIN {X 0,Y 227.895,Z 355.71,A -85,B 0,C 180,E1 -20014.519,E2 -20014.519} C_VEL
LIN {X 0,Y 228.868,Z 358.541,A -85,B 0,C 180,E1 -20015.02,E2 -20015.02} C_VEL
LIN {X 0,Y 230.977,Z 360.721,A -85,B 0,C 180,E1 -20015.804,E2 -20015.804} C_VEL
LIN {X 0,Y 231.703,Z 361.527,A -85,B 0,C 180,E1 -20016.071,E2 -20016.071} C_VEL
LIN {X 0,Y 233.796,Z 364.74,A -85,B 0,C 180,E1 -20016.863,E2 -20016.863} C_VEL
LIN {X 0,Y 235.294,Z 366.459,A -85,B 0,C 180,E1 -20017.387,E2 -20017.387} C_VEL
LIN {X 0,Y 237.992,Z 370.172,A -85,B 0,C 180,E1 -20018.327,E2 -20018.327} C_VEL
LIN {X 0,Y 244.409,Z 379.339,A -85,B 0,C 180,E1 -20020.429,E2 -20020.429} C_VEL
LIN {X 0,Y 249.81,Z 387.85,A -85,B 0,C 180,E1 -20022.088,E2 -20022.088} C_VEL
LIN {X 0,Y 256.924,Z 400.979,A -85,B 0,C 180,E1 -20024.171,E2 -20024.171} C_VEL
LIN {X 0,Y 263.537,Z 415.108,A -85,B 0,C 180,E1 -20026.017,E2 -20026.017} C_VEL
LIN {X 0,Y 263.985,Z 416.418,A -85,B 0,C 180,E1 -20026.149,E2 -20026.149} C_VEL
LIN {X 0,Y 260.226,Z 488.784,A -85,B 0,C 180,E1 -20028.054,E2 -20028.054} C_VEL
LIN {X 0,Y 258.845,Z 502.745,A -85,B 0,C 180,E1 -20028.691,E2 -20028.691} C_VEL
LIN {X 0,Y 256.751,Z 516.389,A -85,B 0,C 180,E1 -20029.579,E2 -20029.579} C_VEL
LIN {X 0,Y 254.141,Z 529.268,A -85,B 0,C 180,E1 -20030.704,E2 -20030.704} C_VEL
LIN {X 0,Y 251.449,Z 541,A -85,B 0,C 180,E1 -20032.055,E2 -20032.055} C_VEL
LIN {X 0,Y 248.127,Z 552.851,A -85,B 0,C 180,E1 -20033.753,E2 -20033.753} C_VEL
LIN {X 0,Y 245.023,Z 562.682,A -85,B 0,C 180,E1 -20035.494,E2 -20035.494} C_VEL
LIN {X 0,Y 241.81,Z 572.288,A -85,B 0,C 180,E1 -20037.594,E2 -20037.594} C_VEL
LIN {X 0,Y 238.569,Z 581.083,A -85,B 0,C 180,E1 -20039.947,E2 -20039.947} C_VEL
LIN {X 0,Y 235.076,Z 589.842,A -85,B 0,C 180,E1 -20042.875,E2 -20042.875} C_VEL
LIN {X 0,Y 232.224,Z 596.89,A -85,B 0,C 180,E1 -20045.885,E2 -20045.885} C_VEL
LIN {X 0,Y 229.631,Z 603.194,A -85,B 0,C 180,E1 -20049.392,E2 -20049.392} C_VEL
LIN {X 0,Y 228.171,Z 606.791,A -85,B 0,C 180,E1 -20052.06,E2 -20052.06} C_VEL
LIN {X 0,Y 226.739,Z 610.291,A -85,B 0,C 180,E1 -20055.643,E2 -20055.643} C_VEL
LIN {X 0,Y 225.889,Z 612.384,A -85,B 0,C 180,E1 -20059.241,E2 -20059.241} C_VEL
LIN {X 0,Y 225.66,Z 613.132,A -85,B 0,C 180,E1 -20062.844,E2 -20062.844} C_VEL
LIN {X 0,Y 225.608,Z 612.829,A -85,B 0,C 180,E1 -20065.458,E2 -20065.458} C_VEL
LIN {X 0,Y 225.714,Z 611.789,A -85,B 0,C 180,E1 -20068.216,E2 -20068.216} C_VEL
LIN {X 0,Y 226.011,Z 609.229,A -85,B 0,C 180,E1 -20071.782,E2 -20071.782} C_VEL
LIN {X 0,Y 226.814,Z 605.247,A -85,B 0,C 180,E1 -20075.334,E2 -20075.334} C_VEL
LIN {X 0,Y 228.264,Z 599.727,A -85,B 0,C 180,E1 -20078.856,E2 -20078.856} C_VEL
LIN {X 0,Y 230.11,Z 592.793,A -85,B 0,C 180,E1 -20082.216,E2 -20082.216} C_VEL
LIN {X 0,Y 231.875,Z 585.775,A -85,B 0,C 180,E1 -20084.93,E2 -20084.93} C_VEL
LIN {X 0,Y 234.309,Z 577.682,A -85,B 0,C 180,E1 -20087.454,E2 -20087.454} C_VEL
LIN {X 0,Y 237.079,Z 567.935,A -85,B 0,C 180,E1 -20089.932,E2 -20089.932} C_VEL
LIN {X 0,Y 239.686,Z 557.136,A -85,B 0,C 180,E1 -20092.18,E2 -20092.18} C_VEL
LIN {X 0,Y 242.513,Z 545.137,A -85,B 0,C 180,E1 -20094.164,E2 -20094.164} C_VEL
LIN {X 0,Y 244.95,Z 533.29,A -85,B 0,C 180,E1 -20095.719,E2 -20095.719} C_VEL
LIN {X 0,Y 247.129,Z 520.273,A -85,B 0,C 180,E1 -20097.066,E2 -20097.066} C_VEL
LIN {X 0,Y 249.095,Z 506.026,A -85,B 0,C 180,E1 -20098.145,E2 -20098.145} C_VEL
LIN {X 0,Y 250.383,Z 491.488,A -85,B 0,C 180,E1 -20098.921,E2 -20098.921} C_VEL
LIN {X 0,Y 251.403,Z 471.897,A -85,B 0,C 180,E1 -20099.528,E2 -20099.528} C_VEL
LIN {X 0,Y 254.18,Z 406.693,A -85,B 0,C 180,E1 -20101.289,E2 -20101.289} C_VEL
LIN {X 0,Y 247.449,Z 390.481,A -85,B 0,C 180,E1 -20102.923,E2 -20102.923} C_VEL
LIN {X 0,Y 242.424,Z 380.156,A -85,B 0,C 180,E1 -20104.161,E2 -20104.161} C_VEL
LIN {X 0,Y 234.645,Z 367.19,A -85,B 0,C 180,E1 -20106.11,E2 -20106.11} C_VEL
LIN {X 0,Y 232.11,Z 363.355,A -85,B 0,C 180,E1 -20106.77,E2 -20106.77} C_VEL
LIN {X 0,Y 230.118,Z 360.09,A -85,B 0,C 180,E1 -20107.313,E2 -20107.313} C_VEL
LIN {X 0,Y 228.446,Z 357.829,A -85,B 0,C 180,E1 -20107.76,E2 -20107.76} C_VEL
LIN {X 0,Y 227.844,Z 355.73,A -85,B 0,C 180,E1 -20108.024,E2 -20108.024} C_VEL
LIN {X 0,Y 227.788,Z 355.733,A -85,B 0,C 180,E1 -20112.748,E2 -20112.748} C_VEL
LIN {X 0,Y 227.787,Z 355.735,A -85,B 0,C 180,E1 -20117.251,E2 -20117.251} C_VEL
LIN {X 0,Y 227.839,Z 355.723,A -85,B 0,C 180,E1 -20121.907,E2 -20121.907} C_VEL
LIN {X 0,Y 227.881,Z 355.715,A -85,B 0,C 180,E1 -20126.378,E2 -20126.378} C_VEL
LIN {X 0,Y 227.873,Z 355.724,A -85,B 0,C 180,E1 -20130.431,E2 -20130.431} C_VEL
LIN {X 0,Y 227.874,Z 355.721,A -85,B 0,C 180,E1 -20134.419,E2 -20134.419} C_VEL
LIN {X 0,Y 227.922,Z 355.689,A -85,B 0,C 180,E1 -20138.282,E2 -20138.282} C_VEL
LIN {X 0,Y 228.012,Z 355.707,A -85,B 0,C 180,E1 -20143.894,E2 -20143.894} C_VEL
LIN {X 0,Y 228.128,Z 355.65,A -85,B 0,C 180,E1 -20149.347,E2 -20149.347} C_VEL
LIN {X 0,Y 228.308,Z 355.67,A -85,B 0,C 180,E1 -20152.927,E2 -20152.927} C_VEL
LIN {X 0,Y 228.548,Z 355.642,A -85,B 0,C 180,E1 -20158.237,E2 -20158.237} C_VEL
LIN {X 0,Y 228.54,Z 355.634,A -85,B 0,C 180,E1 -20161.762,E2 -20161.762} C_VEL
LIN {X 0,Y 228.309,Z 355.669,A -85,B 0,C 180,E1 -20167.072,E2 -20167.072} C_VEL
LIN {X 0,Y 228.148,Z 355.685,A -85,B 0,C 180,E1 -20170.651,E2 -20170.651} C_VEL
LIN {X 0,Y 228.067,Z 355.694,A -85,B 0,C 180,E1 -20174.271,E2 -20174.271} C_VEL
LIN {X 0,Y 228.06,Z 355.703,A -85,B 0,C 180,E1 -20176.105,E2 -20176.105} C_VEL
LIN {X 0,Y 227.323,Z 355.792,A -85,B 0,C 180,E1 -20177.577,E2 -20177.577} C_VEL
LIN {X 0,Y 224.395,Z 356.16,A -85,B 0,C 180,E1 -20179.978,E2 -20179.978} C_VEL
LIN {X 0,Y 221.951,Z 356.458,A -85,B 0,C 180,E1 -20181.936,E2 -20181.936} C_VEL
LIN {X 0,Y 220.924,Z 356.59,A -85,B 0,C 180,E1 -20183.459,E2 -20183.459} C_VEL
LIN {X 0,Y 220.849,Z 356.597,A -85,B 0,C 180,E1 -20183.975,E2 -20183.975} C_VEL
LIN {X 0,Y 220.88,Z 356.597,A -85,B 0,C 180,E1 -20187.012,E2 -20187.012} C_VEL
LIN {X 0,Y 220.819,Z 356.607,A -85,B 0,C 180,E1 -20190.758,E2 -20190.758} C_VEL
LIN {X 0,Y 220.816,Z 356.606,A -85,B 0,C 180,E1 -20194.952,E2 -20194.952} C_VEL
LIN {X 0,Y 220.839,Z 356.607,A -85,B 0,C 180,E1 -20197.287,E2 -20197.287} C_VEL
LIN {X 0,Y 220.776,Z 356.612,A -85,B 0,C 180,E1 -20201.951,E2 -20201.951} C_VEL
LIN {X 0,Y 220.826,Z 356.806,A -85,B 0,C 180,E1 -20203.184,E2 -20203.184} C_VEL
LIN {X 0,Y 222.28,Z 361.788,A -85,B 0,C 180,E1 -20205.668,E2 -20205.668} C_VEL
LIN {X 0,Y 224.966,Z 366.394,A -85,B 0,C 180,E1 -20206.469,E2 -20206.469} C_VEL
LIN {X 0,Y 232.48,Z 380.074,A -85,B 0,C 180,E1 -20208.598,E2 -20208.598} C_VEL
LIN {X 0,Y 239.674,Z 395.351,A -85,B 0,C 180,E1 -20210.54,E2 -20210.54} C_VEL
LIN {X 0,Y 246.469,Z 411.965,A -85,B 0,C 180,E1 -20212.305,E2 -20212.305} C_VEL
LIN {X 0,Y 247.797,Z 423.128,A -85,B 0,C 180,E1 -20212.909,E2 -20212.909} C_VEL
LIN {X 0,Y 244.289,Z 500.206,A -85,B 0,C 180,E1 -20215.062,E2 -20215.062} C_VEL
LIN {X 0,Y 242.793,Z 514.938,A -85,B 0,C 180,E1 -20215.761,E2 -20215.761} C_VEL
LIN {X 0,Y 240.958,Z 528.419,A -85,B 0,C 180,E1 -20216.722,E2 -20216.722} C_VEL
LIN {X 0,Y 238.546,Z 541.575,A -85,B 0,C 180,E1 -20217.973,E2 -20217.973} C_VEL
LIN {X 0,Y 235.792,Z 554.302,A -85,B 0,C 180,E1 -20219.556,E2 -20219.556} C_VEL
LIN {X 0,Y 233.064,Z 565.905,A -85,B 0,C 180,E1 -20221.399,E2 -20221.399} C_VEL
LIN {X 0,Y 230.45,Z 575.549,A -85,B 0,C 180,E1 -20223.267,E2 -20223.267} C_VEL
LIN {X 0,Y 227.391,Z 586.265,A -85,B 0,C 180,E1 -20225.825,E2 -20225.825} C_VEL
LIN {X 0,Y 224.856,Z 595.109,A -85,B 0,C 180,E1 -20228.454,E2 -20228.454} C_VEL
LIN {X 0,Y 222.783,Z 602.505,A -85,B 0,C 180,E1 -20231.153,E2 -20231.153} C_VEL
LIN {X 0,Y 221.505,Z 607.667,A -85,B 0,C 180,E1 -20233.408,E2 -20233.408} C_VEL
LIN {X 0,Y 220.17,Z 612.867,A -85,B 0,C 180,E1 -20236.148,E2 -20236.148} C_VEL
LIN {X 0,Y 219.073,Z 618.312,A -85,B 0,C 180,E1 -20239.837,E2 -20239.837} C_VEL
LIN {X 0,Y 218.675,Z 621.328,A -85,B 0,C 180,E1 -20242.614,E2 -20242.614} C_VEL
LIN {X 0,Y 218.51,Z 624.12,A -85,B 0,C 180,E1 -20246.312,E2 -20246.312} C_VEL
LIN {X 0,Y 218.648,Z 625.53,A -85,B 0,C 180,E1 -20250,E2 -20250} C_VEL
LIN {X 0,Y 218.497,Z 625.579,A -85,B 0,C 180,E1 -20253.689,E2 -20253.689} C_VEL
LIN {X 0,Y 218.679,Z 624.295,A -85,B 0,C 180,E1 -20257.386,E2 -20257.386} C_VEL
LIN {X 0,Y 219.383,Z 621.654,A -85,B 0,C 180,E1 -20261.082,E2 -20261.082} C_VEL
LIN {X 0,Y 220.819,Z 617.585,A -85,B 0,C 180,E1 -20264.751,E2 -20264.751} C_VEL
LIN {X 0,Y 223.019,Z 611.979,A -85,B 0,C 180,E1 -20268.369,E2 -20268.369} C_VEL
LIN {X 0,Y 225.49,Z 605.675,A -85,B 0,C 180,E1 -20271.483,E2 -20271.483} C_VEL
LIN {X 0,Y 228.73,Z 597.849,A -85,B 0,C 180,E1 -20274.507,E2 -20274.507} C_VEL
LIN {X 0,Y 232.006,Z 589.694,A -85,B 0,C 180,E1 -20277.026,E2 -20277.026} C_VEL
LIN {X 0,Y 235.834,Z 579.885,A -85,B 0,C 180,E1 -20279.453,E2 -20279.453} C_VEL
LIN {X 0,Y 239.396,Z 569.622,A -85,B 0,C 180,E1 -20281.511,E2 -20281.511} C_VEL
LIN {X 0,Y 242.886,Z 558.252,A -85,B 0,C 180,E1 -20283.352,E2 -20283.352} C_VEL
LIN {X 0,Y 246.442,Z 545.089,A -85,B 0,C 180,E1 -20285.025,E2 -20285.025} C_VEL
LIN {X 0,Y 249.462,Z 532.035,A -85,B 0,C 180,E1 -20286.273,E2 -20286.273} C_VEL
LIN {X 0,Y 252.051,Z 517.792,A -85,B 0,C 180,E1 -20287.272,E2 -20287.272} C_VEL
LIN {X 0,Y 253.902,Z 503.073,A -85,B 0,C 180,E1 -20287.986,E2 -20287.986} C_VEL
LIN {X 0,Y 255.25,Z 482.536,A -85,B 0,C 180,E1 -20288.588,E2 -20288.588} C_VEL
LIN {X 0,Y 258.119,Z 426.167,A -85,B 0,C 180,E1 -20290.085,E2 -20290.085} C_VEL
LIN {X 0,Y 253.075,Z 413.937,A -85,B 0,C 180,E1 -20291.594,E2 -20291.594} C_VEL
LIN {X 0,Y 246.072,Z 399.48,A -85,B 0,C 180,E1 -20293.761,E2 -20293.761} C_VEL
LIN {X 0,Y 240.193,Z 388.812,A -85,B 0,C 180,E1 -20295.687,E2 -20295.687} C_VEL
LIN {X 0,Y 235.643,Z 381.236,A -85,B 0,C 180,E1 -20297.267,E2 -20297.267} C_VEL
LIN {X 0,Y 232.42,Z 376.132,A -85,B 0,C 180,E1 -20298.444,E2 -20298.444} C_VEL
LIN {X 0,Y 229.325,Z 371.296,A -85,B 0,C 180,E1 -20299.633,E2 -20299.633} C_VEL
LIN {X 0,Y 226.428,Z 366.826,A -85,B 0,C 180,E1 -20300.802,E2 -20300.802} C_VEL
LIN {X 0,Y 222.955,Z 362.137,A -85,B 0,C 180,E1 -20302.253,E2 -20302.253} C_VEL
LIN {X 0,Y 222.152,Z 360.551,A -85,B 0,C 180,E1 -20302.686,E2 -20302.686} C_VEL
LIN {X 0,Y 220.816,Z 356.603,A -85,B 0,C 180,E1 -20305.524,E2 -20305.524} C_VEL
LIN {X 0,Y 220.835,Z 356.596,A -85,B 0,C 180,E1 -20309.39,E2 -20309.39} C_VEL
LIN {X 0,Y 220.877,Z 356.586,A -85,B 0,C 180,E1 -20313.548,E2 -20313.548} C_VEL
LIN {X 0,Y 220.87,Z 356.586,A -85,B 0,C 180,E1 -20317.553,E2 -20317.553} C_VEL
LIN {X 0,Y 220.987,Z 356.57,A -85,B 0,C 180,E1 -20322.572,E2 -20322.572} C_VEL
LIN {X 0,Y 221.015,Z 356.565,A -85,B 0,C 180,E1 -20327.139,E2 -20327.139} C_VEL
LIN {X 0,Y 221.196,Z 356.545,A -85,B 0,C 180,E1 -20330.86,E2 -20330.86} C_VEL
LIN {X 0,Y 221.116,Z 356.567,A -85,B 0,C 180,E1 -20334.529,E2 -20334.529} C_VEL
LIN {X 0,Y 221.473,Z 356.514,A -85,B 0,C 180,E1 -20338.182,E2 -20338.182} C_VEL
LIN {X 0,Y 221.506,Z 356.502,A -85,B 0,C 180,E1 -20341.819,E2 -20341.819} C_VEL
LIN {X 0,Y 221.242,Z 356.535,A -85,B 0,C 180,E1 -20347.301,E2 -20347.301} C_VEL
LIN {X 0,Y 221.062,Z 356.561,A -85,B 0,C 180,E1 -20350.997,E2 -20350.997} C_VEL
LIN {X 0,Y 220.969,Z 356.571,A -85,B 0,C 180,E1 -20356.634,E2 -20356.634} C_VEL
LIN {X 0,Y 220.849,Z 356.588,A -85,B 0,C 180,E1 -20360.491,E2 -20360.491} C_VEL
LIN {X 0,Y 220.798,Z 356.596,A -85,B 0,C 180,E1 -20364.444,E2 -20364.444} C_VEL
LIN {X 0,Y 220.797,Z 356.579,A -85,B 0,C 180,E1 -20368.52,E2 -20368.52} C_VEL
LIN {X 0,Y 220.795,Z 356.6,A -85,B 0,C 180,E1 -20372.085,E2 -20372.085} C_VEL
LIN {X 0,Y 221.547,Z 359.008,A -85,B 0,C 180,E1 -20372.5,E2 -20372.5} C_VEL
LIN {X 0,Y 223.597,Z 361.398,A -85,B 0,C 180,E1 -20373.374,E2 -20373.374} C_VEL
LIN {X 0,Y 224.791,Z 362.346,A -85,B 0,C 180,E1 -20373.844,E2 -20373.844} C_VEL
LIN {X 0,Y 226.821,Z 365.621,A -85,B 0,C 180,E1 -20374.705,E2 -20374.705} C_VEL
LIN {X 0,Y 228.634,Z 367.55,A -85,B 0,C 180,E1 -20375.398,E2 -20375.398} C_VEL
LIN {X 0,Y 231.167,Z 371.042,A -85,B 0,C 180,E1 -20376.368,E2 -20376.368} C_VEL
LIN {X 0,Y 238.329,Z 381.031,A -85,B 0,C 180,E1 -20378.908,E2 -20378.908} C_VEL
LIN {X 0,Y 244.999,Z 391.244,A -85,B 0,C 180,E1 -20381.076,E2 -20381.076} C_VEL
LIN {X 0,Y 252.709,Z 405.708,A -85,B 0,C 180,E1 -20383.447,E2 -20383.447} C_VEL
LIN {X 0,Y 258.557,Z 418.432,A -85,B 0,C 180,E1 -20385.157,E2 -20385.157} C_VEL
LIN {X 0,Y 254.727,Z 489.524,A -85,B 0,C 180,E1 -20387.067,E2 -20387.067} C_VEL
LIN {X 0,Y 253.183,Z 504.073,A -85,B 0,C 180,E1 -20387.756,E2 -20387.756} C_VEL
LIN {X 0,Y 250.913,Z 517.995,A -85,B 0,C 180,E1 -20388.701,E2 -20388.701} C_VEL
LIN {X 0,Y 248.056,Z 531.208,A -85,B 0,C 180,E1 -20389.906,E2 -20389.906} C_VEL
LIN {X 0,Y 245.066,Z 543.521,A -85,B 0,C 180,E1 -20391.409,E2 -20391.409} C_VEL
LIN {X 0,Y 241.611,Z 554.957,A -85,B 0,C 180,E1 -20393.134,E2 -20393.134} C_VEL
LIN {X 0,Y 237.78,Z 566.423,A -85,B 0,C 180,E1 -20395.321,E2 -20395.321} C_VEL
LIN {X 0,Y 234.175,Z 576.614,A -85,B 0,C 180,E1 -20397.811,E2 -20397.811} C_VEL
LIN {X 0,Y 230.718,Z 585.039,A -85,B 0,C 180,E1 -20400.33,E2 -20400.33} C_VEL
LIN {X 0,Y 227.316,Z 593.065,A -85,B 0,C 180,E1 -20403.366,E2 -20403.366} C_VEL
LIN {X 0,Y 224.9,Z 598.693,A -85,B 0,C 180,E1 -20406.031,E2 -20406.031} C_VEL
LIN {X 0,Y 222.314,Z 604.562,A -85,B 0,C 180,E1 -20409.65,E2 -20409.65} C_VEL
LIN {X 0,Y 220.481,Z 608.839,A -85,B 0,C 180,E1 -20413.328,E2 -20413.328} C_VEL
LIN {X 0,Y 219.2,Z 611.658,A -85,B 0,C 180,E1 -20417.03,E2 -20417.03} C_VEL
LIN {X 0,Y 218.65,Z 613.103,A -85,B 0,C 180,E1 -20420.752,E2 -20420.752} C_VEL
LIN {X 0,Y 218.561,Z 613.221,A -85,B 0,C 180,E1 -20424.464,E2 -20424.464} C_VEL
LIN {X 0,Y 218.626,Z 612.03,A -85,B 0,C 180,E1 -20428.158,E2 -20428.158} C_VEL
LIN {X 0,Y 218.946,Z 609.51,A -85,B 0,C 180,E1 -20431.839,E2 -20431.839} C_VEL
LIN {X 0,Y 219.781,Z 605.567,A -85,B 0,C 180,E1 -20435.505,E2 -20435.505} C_VEL
LIN {X 0,Y 221.273,Z 600.084,A -85,B 0,C 180,E1 -20439.138,E2 -20439.138} C_VEL
LIN {X 0,Y 223.047,Z 593.71,A -85,B 0,C 180,E1 -20442.368,E2 -20442.368} C_VEL
LIN {X 0,Y 225.034,Z 586.215,A -85,B 0,C 180,E1 -20445.394,E2 -20445.394} C_VEL
LIN {X 0,Y 227.572,Z 578.17,A -85,B 0,C 180,E1 -20447.989,E2 -20447.989} C_VEL
LIN {X 0,Y 230.45,Z 568.479,A -85,B 0,C 180,E1 -20450.531,E2 -20450.531} C_VEL
LIN {X 0,Y 233.163,Z 557.749,A -85,B 0,C 180,E1 -20452.835,E2 -20452.835} C_VEL
LIN {X 0,Y 236.089,Z 545.836,A -85,B 0,C 180,E1 -20454.865,E2 -20454.865} C_VEL
LIN {X 0,Y 238.626,Z 534.103,A -85,B 0,C 180,E1 -20456.453,E2 -20456.453} C_VEL
LIN {X 0,Y 240.875,Z 521.294,A -85,B 0,C 180,E1 -20457.829,E2 -20457.829} C_VEL
LIN {X 0,Y 242.912,Z 507.402,A -85,B 0,C 180,E1 -20458.928,E2 -20458.928} C_VEL
LIN {X 0,Y 244.254,Z 493.302,A -85,B 0,C 180,E1 -20459.726,E2 -20459.726} C_VEL
LIN {X 0,Y 245.204,Z 477.515,A -85,B 0,C 180,E1 -20460.263,E2 -20460.263} C_VEL
LIN {X 0,Y 248.266,Z 408.651,A -85,B 0,C 180,E1 -20462.155,E2 -20462.155} C_VEL
LIN {X 0,Y 242.057,Z 393.656,A -85,B 0,C 180,E1 -20463.736,E2 -20463.736} C_VEL
LIN {X 0,Y 237.45,Z 384.076,A -85,B 0,C 180,E1 -20464.927,E2 -20464.927} C_VEL
LIN {X 0,Y 228.712,Z 369.416,A -85,B 0,C 180,E1 -20467.235,E2 -20467.235} C_VEL
LIN {X 0,Y 225.407,Z 364.627,A -85,B 0,C 180,E1 -20468.145,E2 -20468.145} C_VEL
LIN {X 0,Y 223.135,Z 361.059,A -85,B 0,C 180,E1 -20468.805,E2 -20468.805} C_VEL
LIN {X 0,Y 221.301,Z 358.533,A -85,B 0,C 180,E1 -20469.338,E2 -20469.338} C_VEL
LIN {X 0,Y 220.796,Z 356.603,A -85,B 0,C 180,E1 -20469.579,E2 -20469.579} C_VEL
LIN {X 0,Y 220.755,Z 356.607,A -85,B 0,C 180,E1 -20474.459,E2 -20474.459} C_VEL
LIN {X 0,Y 220.75,Z 356.606,A -85,B 0,C 180,E1 -20478.042,E2 -20478.042} C_VEL
LIN {X 0,Y 220.827,Z 356.593,A -85,B 0,C 180,E1 -20482.793,E2 -20482.793} C_VEL
LIN {X 0,Y 220.813,Z 356.591,A -85,B 0,C 180,E1 -20487.243,E2 -20487.243} C_VEL
LIN {X 0,Y 220.797,Z 356.597,A -85,B 0,C 180,E1 -20491.48,E2 -20491.48} C_VEL
LIN {X 0,Y 220.806,Z 356.605,A -85,B 0,C 180,E1 -20495.557,E2 -20495.557} C_VEL
LIN {X 0,Y 220.849,Z 356.561,A -85,B 0,C 180,E1 -20499.509,E2 -20499.509} C_VEL
LIN {X 0,Y 220.973,Z 356.583,A -85,B 0,C 180,E1 -20503.366,E2 -20503.366} C_VEL
LIN {X 0,Y 221.053,Z 356.53,A -85,B 0,C 180,E1 -20509.002,E2 -20509.002} C_VEL
LIN {X 0,Y 221.245,Z 356.546,A -85,B 0,C 180,E1 -20512.7,E2 -20512.7} C_VEL
LIN {X 0,Y 221.506,Z 356.518,A -85,B 0,C 180,E1 -20518.181,E2 -20518.181} C_VEL
LIN {X 0,Y 221.473,Z 356.514,A -85,B 0,C 180,E1 -20521.818,E2 -20521.818} C_VEL
LIN {X 0,Y 221.246,Z 356.549,A -85,B 0,C 180,E1 -20527.299,E2 -20527.299} C_VEL
LIN {X 0,Y 221.083,Z 356.567,A -85,B 0,C 180,E1 -20530.995,E2 -20530.995} C_VEL
LIN {X 0,Y 221.019,Z 356.579,A -85,B 0,C 180,E1 -20536.629,E2 -20536.629} C_VEL
LIN {X 0,Y 220.887,Z 356.595,A -85,B 0,C 180,E1 -20540.486,E2 -20540.486} C_VEL
LIN {X 0,Y 220.849,Z 356.597,A -85,B 0,C 180,E1 -20543.975,E2 -20543.975} C_VEL
LIN {X 0,Y 220.207,Z 356.684,A -85,B 0,C 180,E1 -20545.496,E2 -20545.496} C_VEL
LIN {X 0,Y 217.371,Z 357.043,A -85,B 0,C 180,E1 -20547.979,E2 -20547.979} C_VEL
LIN {X 0,Y 214.09,Z 357.446,A -85,B 0,C 180,E1 -20551.051,E2 -20551.051} C_VEL
LIN {X 0,Y 213.74,Z 357.484,A -85,B 0,C 180,E1 -20552.116,E2 -20552.116} C_VEL
LIN {X 0,Y 213.754,Z 357.485,A -85,B 0,C 180,E1 -20556.286,E2 -20556.286} C_VEL
LIN {X 0,Y 213.717,Z 357.493,A -85,B 0,C 180,E1 -20561.124,E2 -20561.124} C_VEL
LIN {X 0,Y 213.738,Z 357.49,A -85,B 0,C 180,E1 -20561.747,E2 -20561.747} C_VEL
LIN {X 0,Y 214.949,Z 361.547,A -85,B 0,C 180,E1 -20563.882,E2 -20563.882} C_VEL
LIN {X 0,Y 217.647,Z 366.12,A -85,B 0,C 180,E1 -20564.757,E2 -20564.757} C_VEL
LIN {X 0,Y 224.078,Z 377.436,A -85,B 0,C 180,E1 -20566.731,E2 -20566.731} C_VEL
LIN {X 0,Y 229.744,Z 388.505,A -85,B 0,C 180,E1 -20568.379,E2 -20568.379} C_VEL
LIN {X 0,Y 235.401,Z 400.924,A -85,B 0,C 180,E1 -20569.962,E2 -20569.962} C_VEL
LIN {X 0,Y 240.985,Z 414.819,A -85,B 0,C 180,E1 -20571.481,E2 -20571.481} C_VEL
LIN {X 0,Y 241.969,Z 423.487,A -85,B 0,C 180,E1 -20571.962,E2 -20571.962} C_VEL
LIN {X 0,Y 238.356,Z 499.676,A -85,B 0,C 180,E1 -20574.125,E2 -20574.125} C_VEL
LIN {X 0,Y 236.936,Z 513.777,A -85,B 0,C 180,E1 -20574.791,E2 -20574.791} C_VEL
LIN {X 0,Y 235.024,Z 527.507,A -85,B 0,C 180,E1 -20575.767,E2 -20575.767} C_VEL
LIN {X 0,Y 232.513,Z 540.818,A -85,B 0,C 180,E1 -20577.039,E2 -20577.039} C_VEL
LIN {X 0,Y 229.656,Z 553.652,A -85,B 0,C 180,E1 -20578.651,E2 -20578.651} C_VEL
LIN {X 0,Y 226.828,Z 565.337,A -85,B 0,C 180,E1 -20580.536,E2 -20580.536} C_VEL
LIN {X 0,Y 224.102,Z 575.044,A -85,B 0,C 180,E1 -20582.447,E2 -20582.447} C_VEL
LIN {X 0,Y 220.872,Z 585.807,A -85,B 0,C 180,E1 -20585.064,E2 -20585.064} C_VEL
LIN {X 0,Y 218.219,Z 594.695,A -85,B 0,C 180,E1 -20587.764,E2 -20587.764} C_VEL
LIN {X 0,Y 215.846,Z 602.705,A -85,B 0,C 180,E1 -20590.776,E2 -20590.776} C_VEL
LIN {X 0,Y 214.147,Z 609.154,A -85,B 0,C 180,E1 -20593.802,E2 -20593.802} C_VEL
LIN {X 0,Y 212.511,Z 615.49,A -85,B 0,C 180,E1 -20597.587,E2 -20597.587} C_VEL
LIN {X 0,Y 211.884,Z 619.106,A -85,B 0,C 180,E1 -20600.454,E2 -20600.454} C_VEL
LIN {X 0,Y 211.484,Z 622.643,A -85,B 0,C 180,E1 -20604.278,E2 -20604.278} C_VEL
LIN {X 0,Y 211.463,Z 624.762,A -85,B 0,C 180,E1 -20608.095,E2 -20608.095} C_VEL
LIN {X 0,Y 211.563,Z 625.31,A -85,B 0,C 180,E1 -20610,E2 -20610} C_VEL
LIN {X 0,Y 211.395,Z 625.383,A -85,B 0,C 180,E1 -20613.813,E2 -20613.813} C_VEL
LIN {X 0,Y 211.619,Z 624.127,A -85,B 0,C 180,E1 -20617.634,E2 -20617.634} C_VEL
LIN {X 0,Y 212.371,Z 621.518,A -85,B 0,C 180,E1 -20621.453,E2 -20621.453} C_VEL
LIN {X 0,Y 213.91,Z 617.479,A -85,B 0,C 180,E1 -20625.239,E2 -20625.239} C_VEL
LIN {X 0,Y 216.242,Z 611.901,A -85,B 0,C 180,E1 -20628.966,E2 -20628.966} C_VEL
LIN {X 0,Y 218.861,Z 605.629,A -85,B 0,C 180,E1 -20632.168,E2 -20632.168} C_VEL
LIN {X 0,Y 222.257,Z 597.839,A -85,B 0,C 180,E1 -20635.27,E2 -20635.27} C_VEL
LIN {X 0,Y 225.695,Z 589.725,A -85,B 0,C 180,E1 -20637.846,E2 -20637.846} C_VEL
LIN {X 0,Y 229.67,Z 579.963,A -85,B 0,C 180,E1 -20640.326,E2 -20640.326} C_VEL
LIN {X 0,Y 233.359,Z 569.757,A -85,B 0,C 180,E1 -20642.424,E2 -20642.424} C_VEL
LIN {X 0,Y 237,Z 558.457,A -85,B 0,C 180,E1 -20644.293,E2 -20644.293} C_VEL
LIN {X 0,Y 240.69,Z 545.385,A -85,B 0,C 180,E1 -20645.99,E2 -20645.99} C_VEL
LIN {X 0,Y 243.804,Z 532.496,A -85,B 0,C 180,E1 -20647.255,E2 -20647.255} C_VEL
LIN {X 0,Y 246.464,Z 518.547,A -85,B 0,C 180,E1 -20648.267,E2 -20648.267} C_VEL
LIN {X 0,Y 248.364,Z 504.353,A -85,B 0,C 180,E1 -20648.988,E2 -20648.988} C_VEL
LIN {X 0,Y 249.609,Z 487.734,A -85,B 0,C 180,E1 -20649.512,E2 -20649.512} C_VEL
LIN {X 0,Y 252.793,Z 428.157,A -85,B 0,C 180,E1 -20651.11,E2 -20651.11} C_VEL
LIN {X 0,Y 246.764,Z 414.079,A -85,B 0,C 180,E1 -20653.003,E2 -20653.003} C_VEL
LIN {X 0,Y 239.95,Z 400.248,A -85,B 0,C 180,E1 -20655.254,E2 -20655.254} C_VEL
LIN {X 0,Y 232.718,Z 387.419,A -85,B 0,C 180,E1 -20657.822,E2 -20657.822} C_VEL
LIN {X 0,Y 226.022,Z 376.793,A -85,B 0,C 180,E1 -20660.425,E2 -20660.425} C_VEL
LIN {X 0,Y 222.407,Z 371.332,A -85,B 0,C 180,E1 -20661.951,E2 -20661.951} C_VEL
LIN {X 0,Y 219.423,Z 366.894,A -85,B 0,C 180,E1 -20663.291,E2 -20663.291} C_VEL
LIN {X 0,Y 215.314,Z 361.455,A -85,B 0,C 180,E1 -20665.239,E2 -20665.239} C_VEL
LIN {X 0,Y 214.718,Z 360.215,A -85,B 0,C 180,E1 -20665.604,E2 -20665.604} C_VEL
LIN {X 0,Y 213.747,Z 357.481,A -85,B 0,C 180,E1 -20667.843,E2 -20667.843} C_VEL
LIN {X 0,Y 213.791,Z 357.475,A -85,B 0,C 180,E1 -20672.599,E2 -20672.599} C_VEL
LIN {X 0,Y 213.813,Z 357.467,A -85,B 0,C 180,E1 -20676.979,E2 -20676.979} C_VEL
LIN {X 0,Y 213.946,Z 357.447,A -85,B 0,C 180,E1 -20682.804,E2 -20682.804} C_VEL
LIN {X 0,Y 213.956,Z 357.443,A -85,B 0,C 180,E1 -20686.707,E2 -20686.707} C_VEL
LIN {X 0,Y 214.136,Z 357.426,A -85,B 0,C 180,E1 -20690.555,E2 -20690.555} C_VEL
LIN {X 0,Y 214.079,Z 357.444,A -85,B 0,C 180,E1 -20694.348,E2 -20694.348} C_VEL
LIN {X 0,Y 214.41,Z 357.393,A -85,B 0,C 180,E1 -20698.122,E2 -20698.122} C_VEL
LIN {X 0,Y 214.516,Z 357.385,A -85,B 0,C 180,E1 -20700.001,E2 -20700.001} C_VEL
LIN {X 0,Y 214.439,Z 357.382,A -85,B 0,C 180,E1 -20701.879,E2 -20701.879} C_VEL
LIN {X 0,Y 214.184,Z 357.415,A -85,B 0,C 180,E1 -20707.543,E2 -20707.543} C_VEL
LIN {X 0,Y 213.991,Z 357.44,A -85,B 0,C 180,E1 -20711.365,E2 -20711.365} C_VEL
LIN {X 0,Y 213.871,Z 357.461,A -85,B 0,C 180,E1 -20715.242,E2 -20715.242} C_VEL
LIN {X 0,Y 213.792,Z 357.476,A -85,B 0,C 180,E1 -20719.192,E2 -20719.192} C_VEL
LIN {X 0,Y 213.766,Z 357.481,A -85,B 0,C 180,E1 -20723.237,E2 -20723.237} C_VEL
LIN {X 0,Y 213.765,Z 357.455,A -85,B 0,C 180,E1 -20728.471,E2 -20728.471} C_VEL
LIN {X 0,Y 213.737,Z 357.473,A -85,B 0,C 180,E1 -20729.283,E2 -20729.283} C_VEL
LIN {X 0,Y 214.587,Z 360.026,A -85,B 0,C 180,E1 -20729.806,E2 -20729.806} C_VEL
LIN {X 0,Y 216.639,Z 362.302,A -85,B 0,C 180,E1 -20730.792,E2 -20730.792} C_VEL
LIN {X 0,Y 217.919,Z 363.309,A -85,B 0,C 180,E1 -20731.361,E2 -20731.361} C_VEL
LIN {X 0,Y 219.776,Z 366.402,A -85,B 0,C 180,E1 -20732.252,E2 -20732.252} C_VEL
LIN {X 0,Y 221.907,Z 368.539,A -85,B 0,C 180,E1 -20733.156,E2 -20733.156} C_VEL
LIN {X 0,Y 224.566,Z 372.227,A -85,B 0,C 180,E1 -20734.287,E2 -20734.287} C_VEL
LIN {X 0,Y 226.088,Z 374.199,A -85,B 0,C 180,E1 -20734.902,E2 -20734.902} C_VEL
LIN {X 0,Y 229.29,Z 378.629,A -85,B 0,C 180,E1 -20736.156,E2 -20736.156} C_VEL
LIN {X 0,Y 235.706,Z 387.798,A -85,B 0,C 180,E1 -20738.489,E2 -20738.489} C_VEL
LIN {X 0,Y 241.118,Z 396.247,A -85,B 0,C 180,E1 -20740.313,E2 -20740.313} C_VEL
LIN {X 0,Y 247.904,Z 409.182,A -85,B 0,C 180,E1 -20742.502,E2 -20742.502} C_VEL
LIN {X 0,Y 253.169,Z 420.567,A -85,B 0,C 180,E1 -20744.118,E2 -20744.118} C_VEL
LIN {X 0,Y 249.424,Z 489.108,A -85,B 0,C 180,E1 -20745.993,E2 -20745.993} C_VEL
LIN {X 0,Y 247.819,Z 503.865,A -85,B 0,C 180,E1 -20746.69,E2 -20746.69} C_VEL
LIN {X 0,Y 245.574,Z 517.323,A -85,B 0,C 180,E1 -20747.598,E2 -20747.598} C_VEL
LIN {X 0,Y 242.575,Z 531.001,A -85,B 0,C 180,E1 -20748.849,E2 -20748.849} C_VEL
LIN {X 0,Y 239.501,Z 543.172,A -85,B 0,C 180,E1 -20750.339,E2 -20750.339} C_VEL
LIN {X 0,Y 235.923,Z 554.706,A -85,B 0,C 180,E1 -20752.091,E2 -20752.091} C_VEL
LIN {X 0,Y 232.605,Z 564.291,A -85,B 0,C 180,E1 -20753.901,E2 -20753.901} C_VEL
LIN {X 0,Y 229.276,Z 573.37,A -85,B 0,C 180,E1 -20756.009,E2 -20756.009} C_VEL
LIN {X 0,Y 225.622,Z 582.32,A -85,B 0,C 180,E1 -20758.55,E2 -20758.55} C_VEL
LIN {X 0,Y 221.834,Z 590.931,A -85,B 0,C 180,E1 -20761.626,E2 -20761.626} C_VEL
LIN {X 0,Y 219.09,Z 596.988,A -85,B 0,C 180,E1 -20764.363,E2 -20764.363} C_VEL
LIN {X 0,Y 216.181,Z 603.323,A -85,B 0,C 180,E1 -20768.046,E2 -20768.046} C_VEL
LIN {X 0,Y 214.501,Z 606.99,A -85,B 0,C 180,E1 -20770.874,E2 -20770.874} C_VEL
LIN {X 0,Y 212.822,Z 610.557,A -85,B 0,C 180,E1 -20774.681,E2 -20774.681} C_VEL
LIN {X 0,Y 211.803,Z 612.713,A -85,B 0,C 180,E1 -20778.516,E2 -20778.516} C_VEL
LIN {X 0,Y 211.487,Z 613.521,A -85,B 0,C 180,E1 -20782.361,E2 -20782.361} C_VEL
LIN {X 0,Y 211.422,Z 613.125,A -85,B 0,C 180,E1 -20785.759,E2 -20785.759} C_VEL
LIN {X 0,Y 211.52,Z 612.271,A -85,B 0,C 180,E1 -20788.096,E2 -20788.096} C_VEL
LIN {X 0,Y 211.861,Z 609.786,A -85,B 0,C 180,E1 -20791.901,E2 -20791.901} C_VEL
LIN {X 0,Y 212.729,Z 605.888,A -85,B 0,C 180,E1 -20795.688,E2 -20795.688} C_VEL
LIN {X 0,Y 214.289,Z 600.44,A -85,B 0,C 180,E1 -20799.438,E2 -20799.438} C_VEL
LIN {X 0,Y 215.998,Z 594.598,A -85,B 0,C 180,E1 -20802.543,E2 -20802.543} C_VEL
LIN {X 0,Y 218.22,Z 586.654,A -85,B 0,C 180,E1 -20805.888,E2 -20805.888} C_VEL
LIN {X 0,Y 220.862,Z 578.657,A -85,B 0,C 180,E1 -20808.555,E2 -20808.555} C_VEL
LIN {X 0,Y 223.849,Z 569.023,A -85,B 0,C 180,E1 -20811.165,E2 -20811.165} C_VEL
LIN {X 0,Y 226.672,Z 558.361,A -85,B 0,C 180,E1 -20813.528,E2 -20813.528} C_VEL
LIN {X 0,Y 229.7,Z 546.533,A -85,B 0,C 180,E1 -20815.606,E2 -20815.606} C_VEL
LIN {X 0,Y 232.344,Z 534.907,A -85,B 0,C 180,E1 -20817.226,E2 -20817.226} C_VEL
LIN {X 0,Y 234.839,Z 521.26,A -85,B 0,C 180,E1 -20818.731,E2 -20818.731} C_VEL
LIN {X 0,Y 236.96,Z 507.25,A -85,B 0,C 180,E1 -20819.849,E2 -20819.849} C_VEL
LIN {X 0,Y 238.353,Z 492.95,A -85,B 0,C 180,E1 -20820.664,E2 -20820.664} C_VEL
LIN {X 0,Y 239.43,Z 474.839,A -85,B 0,C 180,E1 -20821.266,E2 -20821.266} C_VEL
LIN {X 0,Y 242.373,Z 410.368,A -85,B 0,C 180,E1 -20823.078,E2 -20823.078} C_VEL
LIN {X 0,Y 234.822,Z 392.505,A -85,B 0,C 180,E1 -20825.105,E2 -20825.105} C_VEL
LIN {X 0,Y 229.498,Z 382.83,A -85,B 0,C 180,E1 -20826.535,E2 -20826.535} C_VEL
LIN {X 0,Y 223.717,Z 373.389,A -85,B 0,C 180,E1 -20828.156,E2 -20828.156} C_VEL
LIN {X 0,Y 218.698,Z 365.843,A -85,B 0,C 180,E1 -20829.64,E2 -20829.64} C_VEL
LIN {X 0,Y 216.134,Z 361.974,A -85,B 0,C 180,E1 -20830.439,E2 -20830.439} C_VEL
LIN {X 0,Y 214.265,Z 359.495,A -85,B 0,C 180,E1 -20831.025,E2 -20831.025} C_VEL
LIN {X 0,Y 213.699,Z 357.487,A -85,B 0,C 180,E1 -20831.285,E2 -20831.285} C_VEL
LIN {X 0,Y 213.703,Z 357.491,A -85,B 0,C 180,E1 -20833.68,E2 -20833.68} C_VEL
LIN {X 0,Y 213.703,Z 357.489,A -85,B 0,C 180,E1 -20836.345,E2 -20836.345} C_VEL
LIN {X 0,Y 213.704,Z 357.488,A -85,B 0,C 180,E1 -20841.328,E2 -20841.328} C_VEL
LIN {X 0,Y 213.755,Z 357.477,A -85,B 0,C 180,E1 -20846.017,E2 -20846.017} C_VEL
LIN {X 0,Y 213.749,Z 357.483,A -85,B 0,C 180,E1 -20850.448,E2 -20850.448} C_VEL
LIN {X 0,Y 213.753,Z 357.483,A -85,B 0,C 180,E1 -20854.695,E2 -20854.695} C_VEL
LIN {X 0,Y 213.777,Z 357.444,A -85,B 0,C 180,E1 -20858.799,E2 -20858.799} C_VEL
LIN {X 0,Y 213.881,Z 357.459,A -85,B 0,C 180,E1 -20862.798,E2 -20862.798} C_VEL
LIN {X 0,Y 213.919,Z 357.44,A -85,B 0,C 180,E1 -20866.704,E2 -20866.704} C_VEL
LIN {X 0,Y 214.136,Z 357.4,A -85,B 0,C 180,E1 -20870.554,E2 -20870.554} C_VEL
LIN {X 0,Y 214.084,Z 357.442,A -85,B 0,C 180,E1 -20874.347,E2 -20874.347} C_VEL
LIN {X 0,Y 214.439,Z 357.398,A -85,B 0,C 180,E1 -20878.121,E2 -20878.121} C_VEL
LIN {X 0,Y 214.516,Z 357.382,A -85,B 0,C 180,E1 -20879.999,E2 -20879.999} C_VEL
LIN {X 0,Y 214.41,Z 357.394,A -85,B 0,C 180,E1 -20881.878,E2 -20881.878} C_VEL
LIN {X 0,Y 214.187,Z 357.429,A -85,B 0,C 180,E1 -20887.541,E2 -20887.541} C_VEL
LIN {X 0,Y 214.01,Z 357.449,A -85,B 0,C 180,E1 -20891.363,E2 -20891.363} C_VEL
LIN {X 0,Y 213.936,Z 357.457,A -85,B 0,C 180,E1 -20895.236,E2 -20895.236} C_VEL
LIN {X 0,Y 213.839,Z 357.47,A -85,B 0,C 180,E1 -20899.187,E2 -20899.187} C_VEL
LIN {X 0,Y 213.775,Z 357.475,A -85,B 0,C 180,E1 -20903.962,E2 -20903.962} C_VEL
LIN {X 0,Y 213.812,Z 357.479,A -85,B 0,C 180,E1 -20907.44,E2 -20907.44} C_VEL
LIN {X 0,Y 213.74,Z 357.484,A -85,B 0,C 180,E1 -20912.116,E2 -20912.116} C_VEL
LIN {X 0,Y 213.026,Z 357.575,A -85,B 0,C 180,E1 -20913.162,E2 -20913.162} C_VEL
LIN {X 0,Y 210.156,Z 357.934,A -85,B 0,C 180,E1 -20914.806,E2 -20914.806} C_VEL
LIN {X 0,Y 207.317,Z 358.288,A -85,B 0,C 180,E1 -20916.493,E2 -20916.493} C_VEL
LIN {X 0,Y 206.691,Z 358.364,A -85,B 0,C 180,E1 -20917.587,E2 -20917.587} C_VEL
LIN {X 0,Y 206.694,Z 358.566,A -85,B 0,C 180,E1 -20920.389,E2 -20920.389} C_VEL
LIN {X 0,Y 207.464,Z 361.074,A -85,B 0,C 180,E1 -20921.855,E2 -20921.855} C_VEL
LIN {X 0,Y 209.814,Z 365.113,A -85,B 0,C 180,E1 -20922.699,E2 -20922.699} C_VEL
LIN {X 0,Y 211.447,Z 367.746,A -85,B 0,C 180,E1 -20923.259,E2 -20923.259} C_VEL
LIN {X 0,Y 217.363,Z 377.874,A -85,B 0,C 180,E1 -20925.204,E2 -20925.204} C_VEL
LIN {X 0,Y 223.42,Z 389.291,A -85,B 0,C 180,E1 -20927.078,E2 -20927.078} C_VEL
LIN {X 0,Y 229.893,Z 403.534,A -85,B 0,C 180,E1 -20929,E2 -20929} C_VEL
LIN {X 0,Y 235.431,Z 417.427,A -85,B 0,C 180,E1 -20930.588,E2 -20930.588} C_VEL
LIN {X 0,Y 236.149,Z 425.655,A -85,B 0,C 180,E1 -20931.025,E2 -20931.025} C_VEL
LIN {X 0,Y 232.419,Z 500.365,A -85,B 0,C 180,E1 -20933.194,E2 -20933.194} C_VEL
LIN {X 0,Y 230.827,Z 514.907,A -85,B 0,C 180,E1 -20933.917,E2 -20933.917} C_VEL
LIN {X 0,Y 228.965,Z 527.726,A -85,B 0,C 180,E1 -20934.863,E2 -20934.863} C_VEL
LIN {X 0,Y 226.562,Z 540.056,A -85,B 0,C 180,E1 -20936.057,E2 -20936.057} C_VEL
LIN {X 0,Y 223.56,Z 552.994,A -85,B 0,C 180,E1 -20937.695,E2 -20937.695} C_VEL
LIN {X 0,Y 220.641,Z 564.763,A -85,B 0,C 180,E1 -20939.625,E2 -20939.625} C_VEL
LIN {X 0,Y 217.807,Z 574.533,A -85,B 0,C 180,E1 -20941.579,E2 -20941.579} C_VEL
LIN {X 0,Y 214.389,Z 585.346,A -85,B 0,C 180,E1 -20944.256,E2 -20944.256} C_VEL
LIN {X 0,Y 211.597,Z 594.278,A -85,B 0,C 180,E1 -20947.029,E2 -20947.029} C_VEL
LIN {X 0,Y 209.267,Z 601.703,A -85,B 0,C 180,E1 -20949.865,E2 -20949.865} C_VEL
LIN {X 0,Y 207.861,Z 606.975,A -85,B 0,C 180,E1 -20952.284,E2 -20952.284} C_VEL
LIN {X 0,Y 206.324,Z 612.211,A -85,B 0,C 180,E1 -20955.198,E2 -20955.198} C_VEL
LIN {X 0,Y 205.018,Z 617.729,A -85,B 0,C 180,E1 -20959.132,E2 -20959.132} C_VEL
LIN {X 0,Y 204.547,Z 620.785,A -85,B 0,C 180,E1 -20962.101,E2 -20962.101} C_VEL
LIN {X 0,Y 204.335,Z 623.629,A -85,B 0,C 180,E1 -20966.056,E2 -20966.056} C_VEL
LIN {X 0,Y 204.48,Z 625.091,A -85,B 0,C 180,E1 -20970,E2 -20970} C_VEL
LIN {X 0,Y 204.295,Z 625.187,A -85,B 0,C 180,E1 -20973.945,E2 -20973.945} C_VEL
LIN {X 0,Y 204.554,Z 623.957,A -85,B 0,C 180,E1 -20977.899,E2 -20977.899} C_VEL
LIN {X 0,Y 205.378,Z 621.38,A -85,B 0,C 180,E1 -20981.848,E2 -20981.848} C_VEL
LIN {X 0,Y 207.027,Z 617.373,A -85,B 0,C 180,E1 -20985.758,E2 -20985.758} C_VEL
LIN {X 0,Y 209.462,Z 611.825,A -85,B 0,C 180,E1 -20989.605,E2 -20989.605} C_VEL
LIN {X 0,Y 212.267,Z 605.585,A -85,B 0,C 180,E1 -20992.895,E2 -20992.895} C_VEL
LIN {X 0,Y 215.836,Z 597.831,A -85,B 0,C 180,E1 -20996.078,E2 -20996.078} C_VEL
LIN {X 0,Y 219.427,Z 589.757,A -85,B 0,C 180,E1 -20998.714,E2 -20998.714} C_VEL
LIN {X 0,Y 223.566,Z 580.042,A -85,B 0,C 180,E1 -21001.245,E2 -21001.245} C_VEL
LIN {X 0,Y 227.733,Z 568.923,A -85,B 0,C 180,E1 -21003.568,E2 -21003.568} C_VEL
LIN {X 0,Y 231.565,Z 557.374,A -85,B 0,C 180,E1 -21005.482,E2 -21005.482} C_VEL
LIN {X 0,Y 234.997,Z 545.68,A -85,B 0,C 180,E1 -21007.005,E2 -21007.005} C_VEL
LIN {X 0,Y 238.445,Z 531.912,A -85,B 0,C 180,E1 -21008.375,E2 -21008.375} C_VEL
LIN {X 0,Y 241.195,Z 517.785,A -85,B 0,C 180,E1 -21009.396,E2 -21009.396} C_VEL
LIN {X 0,Y 243.099,Z 503.759,A -85,B 0,C 180,E1 -21010.108,E2 -21010.108} C_VEL
LIN {X 0,Y 244.491,Z 485.563,A -85,B 0,C 180,E1 -21010.669,E2 -21010.669} C_VEL
LIN {X 0,Y 247.526,Z 430.401,A -85,B 0,C 180,E1 -21012.175,E2 -21012.175} C_VEL
LIN {X 0,Y 241.528,Z 416.309,A -85,B 0,C 180,E1 -21014.168,E2 -21014.168} C_VEL
LIN {X 0,Y 234.532,Z 402.21,A -85,B 0,C 180,E1 -21016.621,E2 -21016.621} C_VEL
LIN {X 0,Y 228.269,Z 391.194,A -85,B 0,C 180,E1 -21018.983,E2 -21018.983} C_VEL
LIN {X 0,Y 222.647,Z 382.065,A -85,B 0,C 180,E1 -21021.293,E2 -21021.293} C_VEL
LIN {X 0,Y 219.213,Z 376.837,A -85,B 0,C 180,E1 -21022.811,E2 -21022.811} C_VEL
LIN {X 0,Y 215.689,Z 371.576,A -85,B 0,C 180,E1 -21024.479,E2 -21024.479} C_VEL
LIN {X 0,Y 212.318,Z 366.821,A -85,B 0,C 180,E1 -21026.185,E2 -21026.185} C_VEL
LIN {X 0,Y 207.449,Z 360.729,A -85,B 0,C 180,E1 -21028.864,E2 -21028.864} C_VEL
LIN {X 0,Y 207.068,Z 359.802,A -85,B 0,C 180,E1 -21029.158,E2 -21029.158} C_VEL
LIN {X 0,Y 206.712,Z 358.352,A -85,B 0,C 180,E1 -21030.464,E2 -21030.464} C_VEL
LIN {X 0,Y 206.706,Z 358.35,A -85,B 0,C 180,E1 -21033.769,E2 -21033.769} C_VEL
LIN {X 0,Y 206.739,Z 358.345,A -85,B 0,C 180,E1 -21038.042,E2 -21038.042} C_VEL
LIN {X 0,Y 206.876,Z 358.327,A -85,B 0,C 180,E1 -21042.197,E2 -21042.197} C_VEL
LIN {X 0,Y 206.899,Z 358.324,A -85,B 0,C 180,E1 -21046.245,E2 -21046.245} C_VEL
LIN {X 0,Y 207.08,Z 358.308,A -85,B 0,C 180,E1 -21050.231,E2 -21050.231} C_VEL
LIN {X 0,Y 207.042,Z 358.322,A -85,B 0,C 180,E1 -21054.156,E2 -21054.156} C_VEL
LIN {X 0,Y 207.349,Z 358.271,A -85,B 0,C 180,E1 -21058.058,E2 -21058.058} C_VEL
LIN {X 0,Y 207.484,Z 358.261,A -85,B 0,C 180,E1 -21060.001,E2 -21060.001} C_VEL
LIN {X 0,Y 207.376,Z 358.262,A -85,B 0,C 180,E1 -21061.943,E2 -21061.943} C_VEL
LIN {X 0,Y 207.129,Z 358.296,A -85,B 0,C 180,E1 -21067.801,E2 -21067.801} C_VEL
LIN {X 0,Y 206.91,Z 358.321,A -85,B 0,C 180,E1 -21071.76,E2 -21071.76} C_VEL
LIN {X 0,Y 206.804,Z 358.337,A -85,B 0,C 180,E1 -21075.776,E2 -21075.776} C_VEL
LIN {X 0,Y 206.713,Z 358.351,A -85,B 0,C 180,E1 -21079.877,E2 -21079.877} C_VEL
LIN {X 0,Y 206.693,Z 358.354,A -85,B 0,C 180,E1 -21084.082,E2 -21084.082} C_VEL
LIN {X 0,Y 206.702,Z 358.362,A -85,B 0,C 180,E1 -21086.029,E2 -21086.029} C_VEL
LIN {X 0,Y 207.459,Z 360.788,A -85,B 0,C 180,E1 -21086.584,E2 -21086.584} C_VEL
LIN {X 0,Y 209.381,Z 363.043,A -85,B 0,C 180,E1 -21087.671,E2 -21087.671} C_VEL
LIN {X 0,Y 211.071,Z 364.202,A -85,B 0,C 180,E1 -21088.53,E2 -21088.53} C_VEL
LIN {X 0,Y 212.811,Z 367.198,A -85,B 0,C 180,E1 -21089.491,E2 -21089.491} C_VEL
LIN {X 0,Y 215.314,Z 369.757,A -85,B 0,C 180,E1 -21090.699,E2 -21090.699} C_VEL
LIN {X 0,Y 217.818,Z 373.238,A -85,B 0,C 180,E1 -21091.895,E2 -21091.895} C_VEL
LIN {X 0,Y 219.321,Z 374.977,A -85,B 0,C 180,E1 -21092.563,E2 -21092.563} C_VEL
LIN {X 0,Y 223.335,Z 380.411,A -85,B 0,C 180,E1 -21094.296,E2 -21094.296} C_VEL
LIN {X 0,Y 228.701,Z 387.922,A -85,B 0,C 180,E1 -21096.429,E2 -21096.429} C_VEL
LIN {X 0,Y 235.7,Z 398.549,A -85,B 0,C 180,E1 -21098.975,E2 -21098.975} C_VEL
LIN {X 0,Y 241.098,Z 408.481,A -85,B 0,C 180,E1 -21100.831,E2 -21100.831} C_VEL
LIN {X 0,Y 246.363,Z 419.499,A -85,B 0,C 180,E1 -21102.561,E2 -21102.561} C_VEL
LIN {X 0,Y 247.982,Z 423.075,A -85,B 0,C 180,E1 -21103.075,E2 -21103.075} C_VEL
LIN {X 0,Y 244.1,Z 489.854,A -85,B 0,C 180,E1 -21104.92,E2 -21104.92} C_VEL
LIN {X 0,Y 242.435,Z 504.426,A -85,B 0,C 180,E1 -21105.623,E2 -21105.623} C_VEL
LIN {X 0,Y 239.888,Z 518.93,A -85,B 0,C 180,E1 -21106.634,E2 -21106.634} C_VEL
LIN {X 0,Y 237.064,Z 531.154,A -85,B 0,C 180,E1 -21107.777,E2 -21107.777} C_VEL
LIN {X 0,Y 234.014,Z 542.822,A -85,B 0,C 180,E1 -21109.216,E2 -21109.216} C_VEL
LIN {X 0,Y 230.331,Z 554.456,A -85,B 0,C 180,E1 -21110.999,E2 -21110.999} C_VEL
LIN {X 0,Y 227.626,Z 562.154,A -85,B 0,C 180,E1 -21112.426,E2 -21112.426} C_VEL
LIN {X 0,Y 223.561,Z 572.684,A -85,B 0,C 180,E1 -21114.822,E2 -21114.822} C_VEL
LIN {X 0,Y 219.528,Z 582.262,A -85,B 0,C 180,E1 -21117.572,E2 -21117.572} C_VEL
LIN {X 0,Y 215.514,Z 590.918,A -85,B 0,C 180,E1 -21120.715,E2 -21120.715} C_VEL
LIN {X 0,Y 212.492,Z 597.242,A -85,B 0,C 180,E1 -21123.638,E2 -21123.638} C_VEL
LIN {X 0,Y 209.493,Z 603.389,A -85,B 0,C 180,E1 -21127.306,E2 -21127.306} C_VEL
LIN {X 0,Y 207.704,Z 607.091,A -85,B 0,C 180,E1 -21130.222,E2 -21130.222} C_VEL
LIN {X 0,Y 205.889,Z 610.69,A -85,B 0,C 180,E1 -21134.152,E2 -21134.152} C_VEL
LIN {X 0,Y 204.771,Z 612.878,A -85,B 0,C 180,E1 -21138.116,E2 -21138.116} C_VEL
LIN {X 0,Y 204.402,Z 613.716,A -85,B 0,C 180,E1 -21142.095,E2 -21142.095} C_VEL
LIN {X 0,Y 204.349,Z 613.289,A -85,B 0,C 180,E1 -21145.856,E2 -21145.856} C_VEL
LIN {X 0,Y 204.418,Z 612.511,A -85,B 0,C 180,E1 -21148.03,E2 -21148.03} C_VEL
LIN {X 0,Y 204.778,Z 610.059,A -85,B 0,C 180,E1 -21151.967,E2 -21151.967} C_VEL
LIN {X 0,Y 205.681,Z 606.207,A -85,B 0,C 180,E1 -21155.884,E2 -21155.884} C_VEL
LIN {X 0,Y 207.313,Z 600.796,A -85,B 0,C 180,E1 -21159.759,E2 -21159.759} C_VEL
LIN {X 0,Y 208.979,Z 595.41,A -85,B 0,C 180,E1 -21162.764,E2 -21162.764} C_VEL
LIN {X 0,Y 211.077,Z 588.308,A -85,B 0,C 180,E1 -21165.944,E2 -21165.944} C_VEL
LIN {X 0,Y 213.651,Z 580.606,A -85,B 0,C 180,E1 -21168.707,E2 -21168.707} C_VEL
LIN {X 0,Y 216.747,Z 571.328,A -85,B 0,C 180,E1 -21171.394,E2 -21171.394} C_VEL
LIN {X 0,Y 219.683,Z 561.085,A -85,B 0,C 180,E1 -21173.822,E2 -21173.822} C_VEL
LIN {X 0,Y 222.685,Z 549.792,A -85,B 0,C 180,E1 -21175.97,E2 -21175.97} C_VEL
LIN {X 0,Y 225.704,Z 537.286,A -85,B 0,C 180,E1 -21177.845,E2 -21177.845} C_VEL
LIN {X 0,Y 228.183,Z 525.177,A -85,B 0,C 180,E1 -21179.272,E2 -21179.272} C_VEL
LIN {X 0,Y 230.393,Z 511.832,A -85,B 0,C 180,E1 -21180.473,E2 -21180.473} C_VEL
LIN {X 0,Y 232.093,Z 497.461,A -85,B 0,C 180,E1 -21181.411,E2 -21181.411} C_VEL
LIN {X 0,Y 233.187,Z 483.644,A -85,B 0,C 180,E1 -21181.98,E2 -21181.98} C_VEL
LIN {X 0,Y 236.62,Z 412.491,A -85,B 0,C 180,E1 -21184.018,E2 -21184.018} C_VEL
LIN {X 0,Y 229.604,Z 395.843,A -85,B 0,C 180,E1 -21185.999,E2 -21185.999} C_VEL
LIN {X 0,Y 223.677,Z 385.119,A -85,B 0,C 180,E1 -21187.677,E2 -21187.677} C_VEL
LIN {X 0,Y 217.181,Z 374.683,A -85,B 0,C 180,E1 -21189.618,E2 -21189.618} C_VEL
LIN {X 0,Y 212.047,Z 367.092,A -85,B 0,C 180,E1 -21191.252,E2 -21191.252} C_VEL
LIN {X 0,Y 209.95,Z 363.973,A -85,B 0,C 180,E1 -21191.956,E2 -21191.956} C_VEL
LIN {X 0,Y 209.238,Z 362.993,A -85,B 0,C 180,E1 -21192.197,E2 -21192.197} C_VEL
LIN {X 0,Y 207.304,Z 360.579,A -85,B 0,C 180,E1 -21192.852,E2 -21192.852} C_VEL
LIN {X 0,Y 206.676,Z 358.366,A -85,B 0,C 180,E1 -21193.2,E2 -21193.2} C_VEL
LIN {X 0,Y 206.633,Z 358.362,A -85,B 0,C 180,E1 -21198.441,E2 -21198.441} C_VEL
LIN {X 0,Y 206.666,Z 358.357,A -85,B 0,C 180,E1 -21202.256,E2 -21202.256} C_VEL
LIN {X 0,Y 206.702,Z 358.363,A -85,B 0,C 180,E1 -21204.688,E2 -21204.688} C_VEL
LIN {X 0,Y 206.697,Z 358.363,A -85,B 0,C 180,E1 -21209.334,E2 -21209.334} C_VEL
LIN {X 0,Y 206.688,Z 358.354,A -85,B 0,C 180,E1 -21213.765,E2 -21213.765} C_VEL
LIN {X 0,Y 206.715,Z 358.331,A -85,B 0,C 180,E1 -21218.038,E2 -21218.038} C_VEL
LIN {X 0,Y 206.805,Z 358.332,A -85,B 0,C 180,E1 -21222.19,E2 -21222.19} C_VEL
LIN {X 0,Y 206.86,Z 358.327,A -85,B 0,C 180,E1 -21226.241,E2 -21226.241} C_VEL
LIN {X 0,Y 207.08,Z 358.275,A -85,B 0,C 180,E1 -21230.229,E2 -21230.229} C_VEL
LIN {X 0,Y 207.046,Z 358.32,A -85,B 0,C 180,E1 -21234.155,E2 -21234.155} C_VEL
LIN {X 0,Y 207.375,Z 358.277,A -85,B 0,C 180,E1 -21238.057,E2 -21238.057} C_VEL
LIN {X 0,Y 207.484,Z 358.258,A -85,B 0,C 180,E1 -21239.999,E2 -21239.999} C_VEL
LIN {X 0,Y 207.349,Z 358.274,A -85,B 0,C 180,E1 -21241.942,E2 -21241.942} C_VEL
LIN {X 0,Y 207.131,Z 358.31,A -85,B 0,C 180,E1 -21247.8,E2 -21247.8} C_VEL
LIN {X 0,Y 206.934,Z 358.332,A -85,B 0,C 180,E1 -21251.757,E2 -21251.757} C_VEL
LIN {X 0,Y 206.87,Z 358.34,A -85,B 0,C 180,E1 -21255.77,E2 -21255.77} C_VEL
LIN {X 0,Y 206.781,Z 358.352,A -85,B 0,C 180,E1 -21259.869,E2 -21259.869} C_VEL
LIN {X 0,Y 206.748,Z 358.359,A -85,B 0,C 180,E1 -21264.074,E2 -21264.074} C_VEL
LIN {X 0,Y 206.728,Z 358.358,A -85,B 0,C 180,E1 -21268.421,E2 -21268.421} C_VEL
LIN {X 0,Y 206.703,Z 358.361,A -85,B 0,C 180,E1 -21272.956,E2 -21272.956} C_VEL
LIN {X 0,Y 206.723,Z 358.359,A -85,B 0,C 180,E1 -21275.32,E2 -21275.32} C_VEL
LIN {X 0,Y 206.691,Z 358.364,A -85,B 0,C 180,E1 -21277.587,E2 -21277.587} C_VEL
LIN {X 0,Y 206.764,Z 359.054,A -85,B 0,C 180,E1 -21278.625,E2 -21278.625} C_VEL
LIN {X 0,Y 206.927,Z 361.337,A -85,B 0,C 180,E1 -21279.802,E2 -21279.802} C_VEL
LIN {X 0,Y 207.229,Z 364.605,A -85,B 0,C 180,E1 -21280.822,E2 -21280.822} C_VEL
LIN {X 0,Y 207.921,Z 369.411,A -85,B 0,C 180,E1 -21281.889,E2 -21281.889} C_VEL
LIN {X 0,Y 209.768,Z 376.231,A -85,B 0,C 180,E1 -21283.156,E2 -21283.156} C_VEL
LIN {X 0,Y 211.326,Z 379.43,A -85,B 0,C 180,E1 -21283.768,E2 -21283.768} C_VEL
LIN {X 0,Y 216.812,Z 389.546,A -85,B 0,C 180,E1 -21285.583,E2 -21285.583} C_VEL
LIN {X 0,Y 223.846,Z 404.634,A -85,B 0,C 180,E1 -21287.801,E2 -21287.801} C_VEL
LIN {X 0,Y 229.951,Z 420.059,A -85,B 0,C 180,E1 -21289.655,E2 -21289.655} C_VEL
LIN {X 0,Y 230.479,Z 425.842,A -85,B 0,C 180,E1 -21289.98,E2 -21289.98} C_VEL
LIN {X 0,Y 226.632,Z 499.861,A -85,B 0,C 180,E1 -21292.162,E2 -21292.162} C_VEL
LIN {X 0,Y 224.99,Z 514.504,A -85,B 0,C 180,E1 -21292.896,E2 -21292.896} C_VEL
LIN {X 0,Y 222.964,Z 527.945,A -85,B 0,C 180,E1 -21293.911,E2 -21293.911} C_VEL
LIN {X 0,Y 220.289,Z 541.073,A -85,B 0,C 180,E1 -21295.23,E2 -21295.23} C_VEL
LIN {X 0,Y 217.178,Z 553.873,A -85,B 0,C 180,E1 -21296.919,E2 -21296.919} C_VEL
LIN {X 0,Y 214.169,Z 565.372,A -85,B 0,C 180,E1 -21298.879,E2 -21298.879} C_VEL
LIN {X 0,Y 210.913,Z 575.988,A -85,B 0,C 180,E1 -21301.107,E2 -21301.107} C_VEL
LIN {X 0,Y 207.423,Z 586.527,A -85,B 0,C 180,E1 -21303.866,E2 -21303.866} C_VEL
LIN {X 0,Y 204.578,Z 595.228,A -85,B 0,C 180,E1 -21306.73,E2 -21306.73} C_VEL
LIN {X 0,Y 201.979,Z 603.145,A -85,B 0,C 180,E1 -21309.964,E2 -21309.964} C_VEL
LIN {X 0,Y 200.425,Z 608.462,A -85,B 0,C 180,E1 -21312.659,E2 -21312.659} C_VEL
LIN {X 0,Y 198.943,Z 613.419,A -85,B 0,C 180,E1 -21315.683,E2 -21315.683} C_VEL
LIN {X 0,Y 197.792,Z 618.533,A -85,B 0,C 180,E1 -21319.766,E2 -21319.766} C_VEL
LIN {X 0,Y 197.302,Z 622.125,A -85,B 0,C 180,E1 -21323.866,E2 -21323.866} C_VEL
LIN {X 0,Y 197.271,Z 624.297,A -85,B 0,C 180,E1 -21327.958,E2 -21327.958} C_VEL
LIN {X 0,Y 197.379,Z 624.87,A -85,B 0,C 180,E1 -21330,E2 -21330} C_VEL
LIN {X 0,Y 197.205,Z 624.991,A -85,B 0,C 180,E1 -21334.087,E2 -21334.087} C_VEL
LIN {X 0,Y 197.492,Z 623.786,A -85,B 0,C 180,E1 -21338.184,E2 -21338.184} C_VEL
LIN {X 0,Y 198.384,Z 621.238,A -85,B 0,C 180,E1 -21342.272,E2 -21342.272} C_VEL
LIN {X 0,Y 200.167,Z 617.269,A -85,B 0,C 180,E1 -21346.313,E2 -21346.313} C_VEL
LIN {X 0,Y 202.713,Z 611.749,A -85,B 0,C 180,E1 -21350.286,E2 -21350.286} C_VEL
LIN {X 0,Y 205.705,Z 605.542,A -85,B 0,C 180,E1 -21353.669,E2 -21353.669} C_VEL
LIN {X 0,Y 209.453,Z 597.823,A -85,B 0,C 180,E1 -21356.935,E2 -21356.935} C_VEL
LIN {X 0,Y 213.215,Z 589.789,A -85,B 0,C 180,E1 -21359.632,E2 -21359.632} C_VEL
LIN {X 0,Y 217.525,Z 580.12,A -85,B 0,C 180,E1 -21362.215,E2 -21362.215} C_VEL
LIN {X 0,Y 221.609,Z 569.705,A -85,B 0,C 180,E1 -21364.458,E2 -21364.458} C_VEL
LIN {X 0,Y 225.833,Z 557.578,A -85,B 0,C 180,E1 -21366.526,E2 -21366.526} C_VEL
LIN {X 0,Y 229.38,Z 545.978,A -85,B 0,C 180,E1 -21368.07,E2 -21368.07} C_VEL
LIN {X 0,Y 232.95,Z 532.356,A -85,B 0,C 180,E1 -21369.454,E2 -21369.454} C_VEL
LIN {X 0,Y 235.669,Z 519.246,A -85,B 0,C 180,E1 -21370.438,E2 -21370.438} C_VEL
LIN {X 0,Y 237.756,Z 505.071,A -85,B 0,C 180,E1 -21371.197,E2 -21371.197} C_VEL
LIN {X 0,Y 239.077,Z 489.361,A -85,B 0,C 180,E1 -21371.724,E2 -21371.724} C_VEL
LIN {X 0,Y 242.355,Z 432.628,A -85,B 0,C 180,E1 -21373.285,E2 -21373.285} C_VEL
LIN {X 0,Y 236.758,Z 419.518,A -85,B 0,C 180,E1 -21375.246,E2 -21375.246} C_VEL
LIN {X 0,Y 230.344,Z 406.342,A -85,B 0,C 180,E1 -21377.626,E2 -21377.626} C_VEL
LIN {X 0,Y 224.635,Z 396.135,A -85,B 0,C 180,E1 -21379.893,E2 -21379.893} C_VEL
LIN {X 0,Y 219.303,Z 387.315,A -85,B 0,C 180,E1 -21382.197,E2 -21382.197} C_VEL
LIN {X 0,Y 216.124,Z 382.361,A -85,B 0,C 180,E1 -21383.674,E2 -21383.674} C_VEL
LIN {X 0,Y 213.022,Z 377.575,A -85,B 0,C 180,E1 -21385.214,E2 -21385.214} C_VEL
LIN {X 0,Y 208.863,Z 371.772,A -85,B 0,C 180,E1 -21387.427,E2 -21387.427} C_VEL
LIN {X 0,Y 204.815,Z 366.38,A -85,B 0,C 180,E1 -21389.808,E2 -21389.808} C_VEL
LIN {X 0,Y 203.092,Z 364.465,A -85,B 0,C 180,E1 -21390.881,E2 -21390.881} C_VEL
LIN {X 0,Y 200.83,Z 362.316,A -85,B 0,C 180,E1 -21392.354,E2 -21392.354} C_VEL
LIN {X 0,Y 199.766,Z 359.866,A -85,B 0,C 180,E1 -21393.208,E2 -21393.208} C_VEL
LIN {X 0,Y 199.675,Z 359.227,A -85,B 0,C 180,E1 -21393.477,E2 -21393.477} C_VEL
LIN {X 0,Y 199.711,Z 359.222,A -85,B 0,C 180,E1 -21397.226,E2 -21397.226} C_VEL
LIN {X 0,Y 199.798,Z 359.209,A -85,B 0,C 180,E1 -21401.758,E2 -21401.758} C_VEL
LIN {X 0,Y 199.839,Z 359.206,A -85,B 0,C 180,E1 -21405.749,E2 -21405.749} C_VEL
LIN {X 0,Y 200.025,Z 359.191,A -85,B 0,C 180,E1 -21409.882,E2 -21409.882} C_VEL
LIN {X 0,Y 200.006,Z 359.196,A -85,B 0,C 180,E1 -21413.949,E2 -21413.949} C_VEL
LIN {X 0,Y 200.291,Z 359.149,A -85,B 0,C 180,E1 -21417.99,E2 -21417.99} C_VEL
LIN {X 0,Y 200.451,Z 359.136,A -85,B 0,C 180,E1 -21420.001,E2 -21420.001} C_VEL
LIN {X 0,Y 200.315,Z 359.141,A -85,B 0,C 180,E1 -21422.011,E2 -21422.011} C_VEL
LIN {X 0,Y 200.077,Z 359.176,A -85,B 0,C 180,E1 -21428.078,E2 -21428.078} C_VEL
LIN {X 0,Y 199.859,Z 359.2,A -85,B 0,C 180,E1 -21432.181,E2 -21432.181} C_VEL
LIN {X 0,Y 199.744,Z 359.214,A -85,B 0,C 180,E1 -21436.349,E2 -21436.349} C_VEL
LIN {X 0,Y 199.644,Z 359.228,A -85,B 0,C 180,E1 -21440.612,E2 -21440.612} C_VEL
LIN {X 0,Y 199.67,Z 359.231,A -85,B 0,C 180,E1 -21442.098,E2 -21442.098} C_VEL
LIN {X 0,Y 200.477,Z 361.753,A -85,B 0,C 180,E1 -21442.825,E2 -21442.825} C_VEL
LIN {X 0,Y 202.345,Z 363.966,A -85,B 0,C 180,E1 -21444.099,E2 -21444.099} C_VEL
LIN {X 0,Y 204.291,Z 365.197,A -85,B 0,C 180,E1 -21445.265,E2 -21445.265} C_VEL
LIN {X 0,Y 205.938,Z 368.143,A -85,B 0,C 180,E1 -21446.338,E2 -21446.338} C_VEL
LIN {X 0,Y 208.687,Z 370.758,A -85,B 0,C 180,E1 -21447.861,E2 -21447.861} C_VEL
LIN {X 0,Y 211.165,Z 374.25,A -85,B 0,C 180,E1 -21449.217,E2 -21449.217} C_VEL
LIN {X 0,Y 212.798,Z 376.032,A -85,B 0,C 180,E1 -21450.034,E2 -21450.034} C_VEL
LIN {X 0,Y 215.653,Z 379.786,A -85,B 0,C 180,E1 -21451.429,E2 -21451.429} C_VEL
LIN {X 0,Y 220.511,Z 386.443,A -85,B 0,C 180,E1 -21453.629,E2 -21453.629} C_VEL
LIN {X 0,Y 225.644,Z 393.76,A -85,B 0,C 180,E1 -21455.752,E2 -21455.752} C_VEL
LIN {X 0,Y 232.576,Z 404.632,A -85,B 0,C 180,E1 -21458.378,E2 -21458.378} C_VEL
LIN {X 0,Y 238.204,Z 415.452,A -85,B 0,C 180,E1 -21460.391,E2 -21460.391} C_VEL
LIN {X 0,Y 242.801,Z 425.542,A -85,B 0,C 180,E1 -21461.966,E2 -21461.966} C_VEL
LIN {X 0,Y 238.957,Z 489.618,A -85,B 0,C 180,E1 -21463.756,E2 -21463.756} C_VEL
LIN {X 0,Y 237.324,Z 503.641,A -85,B 0,C 180,E1 -21464.422,E2 -21464.422} C_VEL
LIN {X 0,Y 234.974,Z 517.127,A -85,B 0,C 180,E1 -21465.341,E2 -21465.341} C_VEL
LIN {X 0,Y 232.012,Z 529.972,A -85,B 0,C 180,E1 -21466.515,E2 -21466.515} C_VEL
LIN {X 0,Y 229.044,Z 541.038,A -85,B 0,C 180,E1 -21467.839,E2 -21467.839} C_VEL
LIN {X 0,Y 225.211,Z 553.025,A -85,B 0,C 180,E1 -21469.644,E2 -21469.644} C_VEL
LIN {X 0,Y 221.923,Z 561.963,A -85,B 0,C 180,E1 -21471.284,E2 -21471.284} C_VEL
LIN {X 0,Y 218.089,Z 571.631,A -85,B 0,C 180,E1 -21473.483,E2 -21473.483} C_VEL
LIN {X 0,Y 214.166,Z 580.831,A -85,B 0,C 180,E1 -21476.091,E2 -21476.091} C_VEL
LIN {X 0,Y 210.417,Z 588.639,A -85,B 0,C 180,E1 -21478.821,E2 -21478.821} C_VEL
LIN {X 0,Y 206.648,Z 596.164,A -85,B 0,C 180,E1 -21482.161,E2 -21482.161} C_VEL
LIN {X 0,Y 203.619,Z 602.033,A -85,B 0,C 180,E1 -21485.532,E2 -21485.532} C_VEL
LIN {X 0,Y 200.939,Z 607.192,A -85,B 0,C 180,E1 -21489.527,E2 -21489.527} C_VEL
LIN {X 0,Y 198.981,Z 610.824,A -85,B 0,C 180,E1 -21493.587,E2 -21493.587} C_VEL
LIN {X 0,Y 197.747,Z 613.043,A -85,B 0,C 180,E1 -21497.687,E2 -21497.687} C_VEL
LIN {X 0,Y 197.313,Z 613.912,A -85,B 0,C 180,E1 -21501.809,E2 -21501.809} C_VEL
LIN {X 0,Y 197.282,Z 613.851,A -85,B 0,C 180,E1 -21503.865,E2 -21503.865} C_VEL
LIN {X 0,Y 197.318,Z 612.751,A -85,B 0,C 180,E1 -21507.959,E2 -21507.959} C_VEL
LIN {X 0,Y 197.698,Z 610.329,A -85,B 0,C 180,E1 -21512.037,E2 -21512.037} C_VEL
LIN {X 0,Y 198.638,Z 606.518,A -85,B 0,C 180,E1 -21516.093,E2 -21516.093} C_VEL
LIN {X 0,Y 200.346,Z 601.151,A -85,B 0,C 180,E1 -21520.102,E2 -21520.102} C_VEL
LIN {X 0,Y 202.265,Z 595.183,A -85,B 0,C 180,E1 -21523.513,E2 -21523.513} C_VEL
LIN {X 0,Y 204.669,Z 587.524,A -85,B 0,C 180,E1 -21526.97,E2 -21526.97} C_VEL
LIN {X 0,Y 207.503,Z 579.625,A -85,B 0,C 180,E1 -21529.797,E2 -21529.797} C_VEL
LIN {X 0,Y 210.752,Z 570.102,A -85,B 0,C 180,E1 -21532.55,E2 -21532.55} C_VEL
LIN {X 0,Y 213.801,Z 559.576,A -85,B 0,C 180,E1 -21535.038,E2 -21535.038} C_VEL
LIN {X 0,Y 217.056,Z 547.918,A -85,B 0,C 180,E1 -21537.216,E2 -21537.216} C_VEL
LIN {X 0,Y 220.246,Z 534.944,A -85,B 0,C 180,E1 -21539.119,E2 -21539.119} C_VEL
LIN {X 0,Y 222.782,Z 522.193,A -85,B 0,C 180,E1 -21540.577,E2 -21540.577} C_VEL
LIN {X 0,Y 224.954,Z 509.142,A -85,B 0,C 180,E1 -21541.686,E2 -21541.686} C_VEL
LIN {X 0,Y 226.499,Z 495.362,A -85,B 0,C 180,E1 -21542.542,E2 -21542.542} C_VEL
LIN {X 0,Y 227.524,Z 481.19,A -85,B 0,C 180,E1 -21543.085,E2 -21543.085} C_VEL
LIN {X 0,Y 230.906,Z 414.501,A -85,B 0,C 180,E1 -21545.013,E2 -21545.013} C_VEL
LIN {X 0,Y 224.32,Z 398.947,A -85,B 0,C 180,E1 -21546.969,E2 -21546.969} C_VEL
LIN {X 0,Y 217.425,Z 386.545,A -85,B 0,C 180,E1 -21549.04,E2 -21549.04} C_VEL
LIN {X 0,Y 210.583,Z 375.905,A -85,B 0,C 180,E1 -21551.227,E2 -21551.227} C_VEL
LIN {X 0,Y 205.424,Z 368.375,A -85,B 0,C 180,E1 -21553.007,E2 -21553.007} C_VEL
LIN {X 0,Y 203.25,Z 365.301,A -85,B 0,C 180,E1 -21553.797,E2 -21553.797} C_VEL
LIN {X 0,Y 202.68,Z 364.221,A -85,B 0,C 180,E1 -21554.023,E2 -21554.023} C_VEL
LIN {X 0,Y 200.654,Z 362.185,A -85,B 0,C 180,E1 -21554.75,E2 -21554.75} C_VEL
LIN {X 0,Y 199.676,Z 359.827,A -85,B 0,C 180,E1 -21555.182,E2 -21555.182} C_VEL
LIN {X 0,Y 199.595,Z 359.24,A -85,B 0,C 180,E1 -21555.274,E2 -21555.274} C_VEL
LIN {X 0,Y 199.596,Z 359.249,A -85,B 0,C 180,E1 -21560.668,E2 -21560.668} C_VEL
LIN {X 0,Y 199.613,Z 359.241,A -85,B 0,C 180,E1 -21564.076,E2 -21564.076} C_VEL
LIN {X 0,Y 199.688,Z 359.224,A -85,B 0,C 180,E1 -21568.134,E2 -21568.134} C_VEL
LIN {X 0,Y 199.636,Z 359.227,A -85,B 0,C 180,E1 -21572.763,E2 -21572.763} C_VEL
LIN {X 0,Y 199.673,Z 359.22,A -85,B 0,C 180,E1 -21577.221,E2 -21577.221} C_VEL
LIN {X 0,Y 199.747,Z 359.203,A -85,B 0,C 180,E1 -21581.802,E2 -21581.802} C_VEL
LIN {X 0,Y 199.798,Z 359.212,A -85,B 0,C 180,E1 -21585.745,E2 -21585.745} C_VEL
LIN {X 0,Y 200.025,Z 359.15,A -85,B 0,C 180,E1 -21589.881,E2 -21589.881} C_VEL
LIN {X 0,Y 200.009,Z 359.197,A -85,B 0,C 180,E1 -21593.948,E2 -21593.948} C_VEL
LIN {X 0,Y 200.314,Z 359.156,A -85,B 0,C 180,E1 -21597.989,E2 -21597.989} C_VEL
LIN {X 0,Y 200.451,Z 359.134,A -85,B 0,C 180,E1 -21599.999,E2 -21599.999} C_VEL
LIN {X 0,Y 199.996,Z 359.196,A -85,B 0,C 180,E1 -21604.03,E2 -21604.03} C_VEL
LIN {X 0,Y 200.079,Z 359.188,A -85,B 0,C 180,E1 -21608.076,E2 -21608.076} C_VEL
LIN {X 0,Y 199.881,Z 359.213,A -85,B 0,C 180,E1 -21612.178,E2 -21612.178} C_VEL
LIN {X 0,Y 199.807,Z 359.222,A -85,B 0,C 180,E1 -21616.343,E2 -21616.343} C_VEL
LIN {X 0,Y 199.693,Z 359.236,A -85,B 0,C 180,E1 -21620.606,E2 -21620.606} C_VEL
LIN {X 0,Y 199.665,Z 359.236,A -85,B 0,C 180,E1 -21624.985,E2 -21624.985} C_VEL
LIN {X 0,Y 199.629,Z 359.24,A -85,B 0,C 180,E1 -21629.529,E2 -21629.529} C_VEL
LIN {X 0,Y 199.653,Z 359.238,A -85,B 0,C 180,E1 -21632.346,E2 -21632.346} C_VEL
LIN {X 0,Y 199.639,Z 359.242,A -85,B 0,C 180,E1 -21637.601,E2 -21637.601} C_VEL
LIN {X 0,Y 199.663,Z 359.391,A -85,B 0,C 180,E1 -21638.765,E2 -21638.765} C_VEL
LIN {X 0,Y 200.01,Z 360.854,A -85,B 0,C 180,E1 -21639.615,E2 -21639.615} C_VEL
LIN {X 0,Y 202.902,Z 365.459,A -85,B 0,C 180,E1 -21640.744,E2 -21640.744} C_VEL
LIN {X 0,Y 207.495,Z 372.832,A -85,B 0,C 180,E1 -21642.431,E2 -21642.431} C_VEL
LIN {X 0,Y 211.326,Z 379.43,A -85,B 0,C 180,E1 -21643.768,E2 -21643.768} C_VEL
LIN {X 0,Y 212.568,Z 382.755,A -85,B 0,C 180,E1 -21644.239,E2 -21644.239} C_VEL
LIN {X 0,Y 213.251,Z 389.222,A -85,B 0,C 180,E1 -21644.704,E2 -21644.704} C_VEL
LIN {X 0,Y 213.821,Z 395.814,A -85,B 0,C 180,E1 -21645.139,E2 -21645.139} C_VEL
LIN {X 0,Y 214.928,Z 399.333,A -85,B 0,C 180,E1 -21645.563,E2 -21645.563} C_VEL
LIN {X 0,Y 220.675,Z 412.594,A -85,B 0,C 180,E1 -21647.446,E2 -21647.446} C_VEL
LIN {X 0,Y 224.556,Z 422.841,A -85,B 0,C 180,E1 -21648.688,E2 -21648.688} C_VEL
LIN {X 0,Y 224.852,Z 426.645,A -85,B 0,C 180,E1 -21648.902,E2 -21648.902} C_VEL
LIN {X 0,Y 220.924,Z 499.34,A -85,B 0,C 180,E1 -21651.076,E2 -21651.076} C_VEL
LIN {X 0,Y 219.24,Z 514.101,A -85,B 0,C 180,E1 -21651.823,E2 -21651.823} C_VEL
LIN {X 0,Y 217.235,Z 527.025,A -85,B 0,C 180,E1 -21652.801,E2 -21652.801} C_VEL
LIN {X 0,Y 214.446,Z 540.308,A -85,B 0,C 180,E1 -21654.139,E2 -21654.139} C_VEL
LIN {X 0,Y 211.205,Z 553.266,A -85,B 0,C 180,E1 -21655.867,E2 -21655.867} C_VEL
LIN {X 0,Y 208.082,Z 564.796,A -85,B 0,C 180,E1 -21657.862,E2 -21657.862} C_VEL
LIN {X 0,Y 205.357,Z 573.51,A -85,B 0,C 180,E1 -21659.682,E2 -21659.682} C_VEL
LIN {X 0,Y 202.186,Z 582.782,A -85,B 0,C 180,E1 -21662.014,E2 -21662.014} C_VEL
LIN {X 0,Y 198.972,Z 592.073,A -85,B 0,C 180,E1 -21664.921,E2 -21664.921} C_VEL
LIN {X 0,Y 195.87,Z 600.942,A -85,B 0,C 180,E1 -21668.421,E2 -21668.421} C_VEL
LIN {X 0,Y 193.607,Z 608.116,A -85,B 0,C 180,E1 -21672.028,E2 -21672.028} C_VEL
LIN {X 0,Y 192.039,Z 613.104,A -85,B 0,C 180,E1 -21675.157,E2 -21675.157} C_VEL
LIN {X 0,Y 190.769,Z 618.247,A -85,B 0,C 180,E1 -21679.385,E2 -21679.385} C_VEL
LIN {X 0,Y 190.218,Z 621.865,A -85,B 0,C 180,E1 -21683.636,E2 -21683.636} C_VEL
LIN {X 0,Y 190.178,Z 624.064,A -85,B 0,C 180,E1 -21687.882,E2 -21687.882} C_VEL
LIN {X 0,Y 190.281,Z 624.65,A -85,B 0,C 180,E1 -21690,E2 -21690} C_VEL
LIN {X 0,Y 190.126,Z 624.796,A -85,B 0,C 180,E1 -21694.24,E2 -21694.24} C_VEL
LIN {X 0,Y 190.45,Z 623.615,A -85,B 0,C 180,E1 -21698.488,E2 -21698.488} C_VEL
LIN {X 0,Y 191.411,Z 621.094,A -85,B 0,C 180,E1 -21702.727,E2 -21702.727} C_VEL
LIN {X 0,Y 193.332,Z 617.162,A -85,B 0,C 180,E1 -21706.907,E2 -21706.907} C_VEL
LIN {X 0,Y 195.978,Z 611.673,A -85,B 0,C 180,E1 -21711.015,E2 -21711.015} C_VEL
LIN {X 0,Y 199.196,Z 605.498,A -85,B 0,C 180,E1 -21714.492,E2 -21714.492} C_VEL
LIN {X 0,Y 203.137,Z 597.815,A -85,B 0,C 180,E1 -21717.844,E2 -21717.844} C_VEL
LIN {X 0,Y 207.069,Z 589.822,A -85,B 0,C 180,E1 -21720.605,E2 -21720.605} C_VEL
LIN {X 0,Y 211.555,Z 580.201,A -85,B 0,C 180,E1 -21723.24,E2 -21723.24} C_VEL
LIN {X 0,Y 215.576,Z 570.421,A -85,B 0,C 180,E1 -21725.411,E2 -21725.411} C_VEL
LIN {X 0,Y 219.741,Z 559.077,A -85,B 0,C 180,E1 -21727.422,E2 -21727.422} C_VEL
LIN {X 0,Y 223.859,Z 546.281,A -85,B 0,C 180,E1 -21729.185,E2 -21729.185} C_VEL
LIN {X 0,Y 227.295,Z 533.78,A -85,B 0,C 180,E1 -21730.491,E2 -21730.491} C_VEL
LIN {X 0,Y 230.338,Z 519.877,A -85,B 0,C 180,E1 -21731.578,E2 -21731.578} C_VEL
LIN {X 0,Y 232.584,Z 505.452,A -85,B 0,C 180,E1 -21732.376,E2 -21732.376} C_VEL
LIN {X 0,Y 233.964,Z 490.252,A -85,B 0,C 180,E1 -21732.9,E2 -21732.9} C_VEL
LIN {X 0,Y 237.31,Z 435.066,A -85,B 0,C 180,E1 -21734.427,E2 -21734.427} C_VEL
LIN {X 0,Y 231.944,Z 422.318,A -85,B 0,C 180,E1 -21736.424,E2 -21736.424} C_VEL
LIN {X 0,Y 226.041,Z 410.199,A -85,B 0,C 180,E1 -21738.74,E2 -21738.74} C_VEL
LIN {X 0,Y 219.648,Z 398.495,A -85,B 0,C 180,E1 -21741.463,E2 -21741.463} C_VEL
LIN {X 0,Y 213.521,Z 388.48,A -85,B 0,C 180,E1 -21744.349,E2 -21744.349} C_VEL
LIN {X 0,Y 209.97,Z 383.029,A -85,B 0,C 180,E1 -21746.189,E2 -21746.189} C_VEL
LIN {X 0,Y 206.145,Z 377.514,A -85,B 0,C 180,E1 -21748.339,E2 -21748.339} C_VEL
LIN {X 0,Y 202.294,Z 372.128,A -85,B 0,C 180,E1 -21750.737,E2 -21750.737} C_VEL
LIN {X 0,Y 198.802,Z 368.65,A -85,B 0,C 180,E1 -21753.068,E2 -21753.068} C_VEL
LIN {X 0,Y 197.474,Z 365.979,A -85,B 0,C 180,E1 -21754.153,E2 -21754.153} C_VEL
LIN {X 0,Y 194.868,Z 364.413,A -85,B 0,C 180,E1 -21756.121,E2 -21756.121} C_VEL
LIN {X 0,Y 193.107,Z 361.876,A -85,B 0,C 180,E1 -21757.746,E2 -21757.746} C_VEL
LIN {X 0,Y 192.64,Z 360.101,A -85,B 0,C 180,E1 -21758.393,E2 -21758.393} C_VEL
LIN {X 0,Y 192.761,Z 360.086,A -85,B 0,C 180,E1 -21763.042,E2 -21763.042} C_VEL
LIN {X 0,Y 192.808,Z 360.078,A -85,B 0,C 180,E1 -21767.368,E2 -21767.368} C_VEL
LIN {X 0,Y 193.027,Z 360.049,A -85,B 0,C 180,E1 -21771.626,E2 -21771.626} C_VEL
LIN {X 0,Y 193.235,Z 360.027,A -85,B 0,C 180,E1 -21777.916,E2 -21777.916} C_VEL
LIN {X 0,Y 193.418,Z 360.012,A -85,B 0,C 180,E1 -21780.001,E2 -21780.001} C_VEL
LIN {X 0,Y 192.959,Z 360.075,A -85,B 0,C 180,E1 -21784.178,E2 -21784.178} C_VEL
LIN {X 0,Y 193.028,Z 360.057,A -85,B 0,C 180,E1 -21788.375,E2 -21788.375} C_VEL
LIN {X 0,Y 192.784,Z 360.083,A -85,B 0,C 180,E1 -21792.635,E2 -21792.635} C_VEL
LIN {X 0,Y 192.719,Z 360.271,A -85,B 0,C 180,E1 -21797.199,E2 -21797.199} C_VEL
LIN {X 0,Y 193.344,Z 362.299,A -85,B 0,C 180,E1 -21797.929,E2 -21797.929} C_VEL
LIN {X 0,Y 195.047,Z 364.633,A -85,B 0,C 180,E1 -21799.47,E2 -21799.47} C_VEL
LIN {X 0,Y 197.583,Z 366.273,A -85,B 0,C 180,E1 -21801.383,E2 -21801.383} C_VEL
LIN {X 0,Y 199.16,Z 369.165,A -85,B 0,C 180,E1 -21802.636,E2 -21802.636} C_VEL
LIN {X 0,Y 202.217,Z 372.02,A -85,B 0,C 180,E1 -21804.65,E2 -21804.65} C_VEL
LIN {X 0,Y 204.521,Z 375.321,A -85,B 0,C 180,E1 -21806.127,E2 -21806.127} C_VEL
LIN {X 0,Y 206.383,Z 377.168,A -85,B 0,C 180,E1 -21807.192,E2 -21807.192} C_VEL
LIN {X 0,Y 209.263,Z 380.956,A -85,B 0,C 180,E1 -21808.799,E2 -21808.799} C_VEL
LIN {X 0,Y 210.893,Z 383.22,A -85,B 0,C 180,E1 -21809.666,E2 -21809.666} C_VEL
LIN {X 0,Y 214.116,Z 387.414,A -85,B 0,C 180,E1 -21811.265,E2 -21811.265} C_VEL
LIN {X 0,Y 219.238,Z 394.529,A -85,B 0,C 180,E1 -21813.613,E2 -21813.613} C_VEL
LIN {X 0,Y 226.447,Z 405.599,A -85,B 0,C 180,E1 -21816.597,E2 -21816.597} C_VEL
LIN {X 0,Y 230.941,Z 413.47,A -85,B 0,C 180,E1 -21818.321,E2 -21818.321} C_VEL
LIN {X 0,Y 237.236,Z 426.81,A -85,B 0,C 180,E1 -21820.634,E2 -21820.634} C_VEL
LIN {X 0,Y 237.733,Z 428.033,A -85,B 0,C 180,E1 -21820.815,E2 -21820.815} C_VEL
LIN {X 0,Y 233.846,Z 490.018,A -85,B 0,C 180,E1 -21822.567,E2 -21822.567} C_VEL
LIN {X 0,Y 232.119,Z 504.262,A -85,B 0,C 180,E1 -21823.258,E2 -21823.258} C_VEL
LIN {X 0,Y 229.434,Z 518.742,A -85,B 0,C 180,E1 -21824.273,E2 -21824.273} C_VEL
LIN {X 0,Y 226.34,Z 531.456,A -85,B 0,C 180,E1 -21825.481,E2 -21825.481} C_VEL
LIN {X 0,Y 223.324,Z 542.132,A -85,B 0,C 180,E1 -21826.805,E2 -21826.805} C_VEL
LIN {X 0,Y 219.359,Z 553.96,A -85,B 0,C 180,E1 -21828.639,E2 -21828.639} C_VEL
LIN {X 0,Y 215.577,Z 563.772,A -85,B 0,C 180,E1 -21830.526,E2 -21830.526} C_VEL
LIN {X 0,Y 211.317,Z 573.862,A -85,B 0,C 180,E1 -21832.959,E2 -21832.959} C_VEL
LIN {X 0,Y 206.849,Z 583.504,A -85,B 0,C 180,E1 -21835.902,E2 -21835.902} C_VEL
LIN {X 0,Y 202.486,Z 592.012,A -85,B 0,C 180,E1 -21839.206,E2 -21839.206} C_VEL
LIN {X 0,Y 198.855,Z 598.84,A -85,B 0,C 180,E1 -21842.648,E2 -21842.648} C_VEL
LIN {X 0,Y 196.255,Z 603.521,A -85,B 0,C 180,E1 -21845.68,E2 -21845.68} C_VEL
LIN {X 0,Y 193.623,Z 608.353,A -85,B 0,C 180,E1 -21849.829,E2 -21849.829} C_VEL
LIN {X 0,Y 192.103,Z 610.957,A -85,B 0,C 180,E1 -21852.982,E2 -21852.982} C_VEL
LIN {X 0,Y 190.736,Z 613.208,A -85,B 0,C 180,E1 -21857.227,E2 -21857.227} C_VEL
LIN {X 0,Y 190.223,Z 614.107,A -85,B 0,C 180,E1 -21861.501,E2 -21861.501} C_VEL
LIN {X 0,Y 190.192,Z 614.061,A -85,B 0,C 180,E1 -21863.635,E2 -21863.635} C_VEL
LIN {X 0,Y 190.222,Z 612.991,A -85,B 0,C 180,E1 -21867.883,E2 -21867.883} C_VEL
LIN {X 0,Y 190.62,Z 610.599,A -85,B 0,C 180,E1 -21872.113,E2 -21872.113} C_VEL
LIN {X 0,Y 191.6,Z 606.825,A -85,B 0,C 180,E1 -21876.318,E2 -21876.318} C_VEL
LIN {X 0,Y 193.388,Z 601.505,A -85,B 0,C 180,E1 -21880.469,E2 -21880.469} C_VEL
LIN {X 0,Y 195.098,Z 596.425,A -85,B 0,C 180,E1 -21883.54,E2 -21883.54} C_VEL
LIN {X 0,Y 197.496,Z 589.159,A -85,B 0,C 180,E1 -21887.072,E2 -21887.072} C_VEL
LIN {X 0,Y 200.331,Z 581.527,A -85,B 0,C 180,E1 -21890.002,E2 -21890.002} C_VEL
LIN {X 0,Y 203.664,Z 572.369,A -85,B 0,C 180,E1 -21892.843,E2 -21892.843} C_VEL
LIN {X 0,Y 206.859,Z 562.276,A -85,B 0,C 180,E1 -21895.4,E2 -21895.4} C_VEL
LIN {X 0,Y 210.075,Z 551.174,A -85,B 0,C 180,E1 -21897.658,E2 -21897.658} C_VEL
LIN {X 0,Y 213.319,Z 538.892,A -85,B 0,C 180,E1 -21899.616,E2 -21899.616} C_VEL
LIN {X 0,Y 215.997,Z 527.087,A -85,B 0,C 180,E1 -21901.1,E2 -21901.1} C_VEL
LIN {X 0,Y 218.356,Z 514.21,A -85,B 0,C 180,E1 -21902.35,E2 -21902.35} C_VEL
LIN {X 0,Y 220.243,Z 500.455,A -85,B 0,C 180,E1 -21903.326,E2 -21903.326} C_VEL
LIN {X 0,Y 221.52,Z 486.334,A -85,B 0,C 180,E1 -21903.989,E2 -21903.989} C_VEL
LIN {X 0,Y 225.216,Z 416.539,A -85,B 0,C 180,E1 -21906.068,E2 -21906.068} C_VEL
LIN {X 0,Y 219.249,Z 402.283,A -85,B 0,C 180,E1 -21907.942,E2 -21907.942} C_VEL
LIN {X 0,Y 211.526,Z 388.641,A -85,B 0,C 180,E1 -21910.396,E2 -21910.396} C_VEL
LIN {X 0,Y 204.305,Z 377.53,A -85,B 0,C 180,E1 -21912.877,E2 -21912.877} C_VEL
LIN {X 0,Y 200.711,Z 372.472,A -85,B 0,C 180,E1 -21914.199,E2 -21914.199} C_VEL
LIN {X 0,Y 198.822,Z 369.64,A -85,B 0,C 180,E1 -21914.937,E2 -21914.937} C_VEL
LIN {X 0,Y 196.36,Z 366.32,A -85,B 0,C 180,E1 -21915.915,E2 -21915.915} C_VEL
LIN {X 0,Y 195.599,Z 365.112,A -85,B 0,C 180,E1 -21916.236,E2 -21916.236} C_VEL
LIN {X 0,Y 193.485,Z 362.918,A -85,B 0,C 180,E1 -21917.088,E2 -21917.088} C_VEL
LIN {X 0,Y 192.58,Z 360.467,A -85,B 0,C 180,E1 -21917.549,E2 -21917.549} C_VEL
LIN {X 0,Y 192.539,Z 360.121,A -85,B 0,C 180,E1 -21917.655,E2 -21917.655} C_VEL
LIN {X 0,Y 192.583,Z 360.112,A -85,B 0,C 180,E1 -21923.404,E2 -21923.404} C_VEL
LIN {X 0,Y 192.607,Z 360.104,A -85,B 0,C 180,E1 -21927.061,E2 -21927.061} C_VEL
LIN {X 0,Y 192.621,Z 360.103,A -85,B 0,C 180,E1 -21931.684,E2 -21931.684} C_VEL
LIN {X 0,Y 192.664,Z 360.106,A -85,B 0,C 180,E1 -21936.342,E2 -21936.342} C_VEL
LIN {X 0,Y 192.696,Z 360.076,A -85,B 0,C 180,E1 -21941.491,E2 -21941.491} C_VEL
LIN {X 0,Y 192.725,Z 360.1,A -85,B 0,C 180,E1 -21945.21,E2 -21945.21} C_VEL
LIN {X 0,Y 192.947,Z 360.029,A -85,B 0,C 180,E1 -21949.566,E2 -21949.566} C_VEL
LIN {X 0,Y 192.973,Z 360.073,A -85,B 0,C 180,E1 -21953.727,E2 -21953.727} C_VEL
LIN {X 0,Y 193.256,Z 360.035,A -85,B 0,C 180,E1 -21957.915,E2 -21957.915} C_VEL
LIN {X 0,Y 193.417,Z 360.01,A -85,B 0,C 180,E1 -21959.999,E2 -21959.999} C_VEL
LIN {X 0,Y 192.943,Z 360.073,A -85,B 0,C 180,E1 -21964.177,E2 -21964.177} C_VEL
LIN {X 0,Y 193.029,Z 360.065,A -85,B 0,C 180,E1 -21968.374,E2 -21968.374} C_VEL
LIN {X 0,Y 192.807,Z 360.093,A -85,B 0,C 180,E1 -21972.632,E2 -21972.632} C_VEL
LIN {X 0,Y 192.76,Z 360.099,A -85,B 0,C 180,E1 -21976.958,E2 -21976.958} C_VEL
LIN {X 0,Y 192.623,Z 360.112,A -85,B 0,C 180,E1 -21981.398,E2 -21981.398} C_VEL
LIN {X 0,Y 192.648,Z 360.114,A -85,B 0,C 180,E1 -21984.213,E2 -21984.213} C_VEL
LIN {X 0,Y 192.629,Z 360.112,A -85,B 0,C 180,E1 -21988.88,E2 -21988.88} C_VEL
LIN {X 0,Y 192.597,Z 360.119,A -85,B 0,C 180,E1 -21993.186,E2 -21993.186} C_VEL
LIN {X 0,Y 192.627,Z 360.296,A -85,B 0,C 180,E1 -21997.012,E2 -21997.012} C_VEL
LIN {X 0,Y 193.829,Z 363.318,A -85,B 0,C 180,E1 -21997.694,E2 -21997.694} C_VEL
LIN {X 0,Y 196.351,Z 366.184,A -85,B 0,C 180,E1 -21998.712,E2 -21998.712} C_VEL
LIN {X 0,Y 203.367,Z 377.497,A -85,B 0,C 180,E1 -22001.487,E2 -22001.487} C_VEL
LIN {X 0,Y 210.297,Z 389.938,A -85,B 0,C 180,E1 -22003.987,E2 -22003.987} C_VEL
LIN {X 0,Y 214.928,Z 399.333,A -85,B 0,C 180,E1 -22005.563,E2 -22005.563} C_VEL
LIN {X 0,Y 216.94,Z 404.334,A -85,B 0,C 180,E1 -22006.255,E2 -22006.255} C_VEL
LIN {X 0,Y 218.642,Z 411.68,A -85,B 0,C 180,E1 -22006.958,E2 -22006.958} C_VEL
LIN {X 0,Y 219.279,Z 417.512,A -85,B 0,C 180,E1 -22007.345,E2 -22007.345} C_VEL
LIN {X 0,Y 219.408,Z 425.491,A -85,B 0,C 180,E1 -22007.708,E2 -22007.708} C_VEL
LIN {X 0,Y 219.203,Z 429.512,A -85,B 0,C 180,E1 -22007.832,E2 -22007.832} C_VEL
LIN {X 0,Y 215.208,Z 499.98,A -85,B 0,C 180,E1 -22009.989,E2 -22009.989} C_VEL
LIN {X 0,Y 213.457,Z 514.452,A -85,B 0,C 180,E1 -22010.745,E2 -22010.745} C_VEL
LIN {X 0,Y 211.379,Z 527.233,A -85,B 0,C 180,E1 -22011.738,E2 -22011.738} C_VEL
LIN {X 0,Y 208.694,Z 539.536,A -85,B 0,C 180,E1 -22012.989,E2 -22012.989} C_VEL
LIN {X 0,Y 205.308,Z 552.602,A -85,B 0,C 180,E1 -22014.744,E2 -22014.744} C_VEL
LIN {X 0,Y 201.725,Z 565.311,A -85,B 0,C 180,E1 -22016.996,E2 -22016.996} C_VEL
LIN {X 0,Y 199.194,Z 572.993,A -85,B 0,C 180,E1 -22018.64,E2 -22018.64} C_VEL
LIN {X 0,Y 195.302,Z 583.963,A -85,B 0,C 180,E1 -22021.523,E2 -22021.523} C_VEL
LIN {X 0,Y 191.975,Z 593.021,A -85,B 0,C 180,E1 -22024.523,E2 -22024.523} C_VEL
LIN {X 0,Y 188.829,Z 601.691,A -85,B 0,C 180,E1 -22028.149,E2 -22028.149} C_VEL
LIN {X 0,Y 186.815,Z 607.769,A -85,B 0,C 180,E1 -22031.351,E2 -22031.351} C_VEL
LIN {X 0,Y 185.152,Z 612.789,A -85,B 0,C 180,E1 -22034.591,E2 -22034.591} C_VEL
LIN {X 0,Y 183.763,Z 617.96,A -85,B 0,C 180,E1 -22038.976,E2 -22038.976} C_VEL
LIN {X 0,Y 183.134,Z 621.605,A -85,B 0,C 180,E1 -22043.389,E2 -22043.389} C_VEL
LIN {X 0,Y 183.052,Z 623.384,A -85,B 0,C 180,E1 -22046.586,E2 -22046.586} C_VEL
LIN {X 0,Y 183.185,Z 624.429,A -85,B 0,C 180,E1 -22050,E2 -22050} C_VEL
LIN {X 0,Y 183.033,Z 624.6,A -85,B 0,C 180,E1 -22054.404,E2 -22054.404} C_VEL
LIN {X 0,Y 183.399,Z 623.444,A -85,B 0,C 180,E1 -22058.817,E2 -22058.817} C_VEL
LIN {X 0,Y 184.435,Z 620.948,A -85,B 0,C 180,E1 -22063.217,E2 -22063.217} C_VEL
LIN {X 0,Y 186.518,Z 617.052,A -85,B 0,C 180,E1 -22067.544,E2 -22067.544} C_VEL
LIN {X 0,Y 189.298,Z 611.598,A -85,B 0,C 180,E1 -22071.794,E2 -22071.794} C_VEL
LIN {X 0,Y 192.18,Z 606.433,A -85,B 0,C 180,E1 -22074.87,E2 -22074.87} C_VEL
LIN {X 0,Y 196.212,Z 599.035,A -85,B 0,C 180,E1 -22078.333,E2 -22078.333} C_VEL
LIN {X 0,Y 200.991,Z 589.857,A -85,B 0,C 180,E1 -22081.635,E2 -22081.635} C_VEL
LIN {X 0,Y 205.649,Z 580.284,A -85,B 0,C 180,E1 -22084.325,E2 -22084.325} C_VEL
LIN {X 0,Y 210.032,Z 570.039,A -85,B 0,C 180,E1 -22086.639,E2 -22086.639} C_VEL
LIN {X 0,Y 214.597,Z 558.001,A -85,B 0,C 180,E1 -22088.781,E2 -22088.781} C_VEL
LIN {X 0,Y 218.424,Z 546.584,A -85,B 0,C 180,E1 -22090.357,E2 -22090.357} C_VEL
LIN {X 0,Y 221.973,Z 534.212,A -85,B 0,C 180,E1 -22091.675,E2 -22091.675} C_VEL
LIN {X 0,Y 225.104,Z 520.505,A -85,B 0,C 180,E1 -22092.771,E2 -22092.771} C_VEL
LIN {X 0,Y 227.409,Z 506.514,A -85,B 0,C 180,E1 -22093.573,E2 -22093.573} C_VEL
LIN {X 0,Y 228.842,Z 492.51,A -85,B 0,C 180,E1 -22094.092,E2 -22094.092} C_VEL
LIN {X 0,Y 232.32,Z 437.412,A -85,B 0,C 180,E1 -22095.635,E2 -22095.635} C_VEL
LIN {X 0,Y 227.185,Z 425.157,A -85,B 0,C 180,E1 -22097.664,E2 -22097.664} C_VEL
LIN {X 0,Y 221.761,Z 413.907,A -85,B 0,C 180,E1 -22099.927,E2 -22099.927} C_VEL
LIN {X 0,Y 216.485,Z 404.009,A -85,B 0,C 180,E1 -22102.304,E2 -22102.304} C_VEL
LIN {X 0,Y 210.526,Z 394.001,A -85,B 0,C 180,E1 -22105.256,E2 -22105.256} C_VEL
LIN {X 0,Y 206.932,Z 388.408,A -85,B 0,C 180,E1 -22107.22,E2 -22107.22} C_VEL
LIN {X 0,Y 203.723,Z 383.589,A -85,B 0,C 180,E1 -22109.126,E2 -22109.126} C_VEL
LIN {X 0,Y 199.505,Z 377.753,A -85,B 0,C 180,E1 -22111.89,E2 -22111.89} C_VEL
LIN {X 0,Y 196.859,Z 375.061,A -85,B 0,C 180,E1 -22113.755,E2 -22113.755} C_VEL
LIN {X 0,Y 195.481,Z 372.646,A -85,B 0,C 180,E1 -22114.898,E2 -22114.898} C_VEL
LIN {X 0,Y 192.947,Z 370.723,A -85,B 0,C 180,E1 -22116.949,E2 -22116.949} C_VEL
LIN {X 0,Y 191.169,Z 367.893,A -85,B 0,C 180,E1 -22118.714,E2 -22118.714} C_VEL
LIN {X 0,Y 190.711,Z 366.938,A -85,B 0,C 180,E1 -22119.226,E2 -22119.226} C_VEL
LIN {X 0,Y 187.788,Z 365.184,A -85,B 0,C 180,E1 -22122.342,E2 -22122.342} C_VEL
LIN {X 0,Y 186.16,Z 362.733,A -85,B 0,C 180,E1 -22124.677,E2 -22124.677} C_VEL
LIN {X 0,Y 185.709,Z 360.967,A -85,B 0,C 180,E1 -22125.621,E2 -22125.621} C_VEL
LIN {X 0,Y 185.89,Z 360.956,A -85,B 0,C 180,E1 -22129.42,E2 -22129.42} C_VEL
LIN {X 0,Y 185.934,Z 360.943,A -85,B 0,C 180,E1 -22133.49,E2 -22133.49} C_VEL
LIN {X 0,Y 186.181,Z 360.905,A -85,B 0,C 180,E1 -22137.837,E2 -22137.837} C_VEL
LIN {X 0,Y 186.383,Z 360.887,A -85,B 0,C 180,E1 -22140.001,E2 -22140.001} C_VEL
LIN {X 0,Y 185.906,Z 360.954,A -85,B 0,C 180,E1 -22144.337,E2 -22144.337} C_VEL
LIN {X 0,Y 185.977,Z 360.938,A -85,B 0,C 180,E1 -22148.695,E2 -22148.695} C_VEL
LIN {X 0,Y 185.946,Z 361.154,A -85,B 0,C 180,E1 -22150.203,E2 -22150.203} C_VEL
LIN {X 0,Y 186.577,Z 363.395,A -85,B 0,C 180,E1 -22151.407,E2 -22151.407} C_VEL
LIN {X 0,Y 188.342,Z 365.682,A -85,B 0,C 180,E1 -22153.762,E2 -22153.762} C_VEL
LIN {X 0,Y 190.939,Z 367.133,A -85,B 0,C 180,E1 -22156.438,E2 -22156.438} C_VEL
LIN {X 0,Y 192.502,Z 370.251,A -85,B 0,C 180,E1 -22158.09,E2 -22158.09} C_VEL
LIN {X 0,Y 195.019,Z 372.405,A -85,B 0,C 180,E1 -22160.193,E2 -22160.193} C_VEL
LIN {X 0,Y 195.712,Z 373.053,A -85,B 0,C 180,E1 -22160.736,E2 -22160.736} C_VEL
LIN {X 0,Y 197.756,Z 376.228,A -85,B 0,C 180,E1 -22162.358,E2 -22162.358} C_VEL
LIN {X 0,Y 200.046,Z 378.325,A -85,B 0,C 180,E1 -22163.911,E2 -22163.911} C_VEL
LIN {X 0,Y 202.339,Z 381.632,A -85,B 0,C 180,E1 -22165.443,E2 -22165.443} C_VEL
LIN {X 0,Y 204.132,Z 383.578,A -85,B 0,C 180,E1 -22166.52,E2 -22166.52} C_VEL
LIN {X 0,Y 207.873,Z 388.568,A -85,B 0,C 180,E1 -22168.664,E2 -22168.664} C_VEL
LIN {X 0,Y 211.523,Z 393.568,A -85,B 0,C 180,E1 -22170.575,E2 -22170.575} C_VEL
LIN {X 0,Y 216.292,Z 400.37,A -85,B 0,C 180,E1 -22172.857,E2 -22172.857} C_VEL
LIN {X 0,Y 223.111,Z 411.062,A -85,B 0,C 180,E1 -22175.808,E2 -22175.808} C_VEL
LIN {X 0,Y 227.287,Z 418.665,A -85,B 0,C 180,E1 -22177.492,E2 -22177.492} C_VEL
LIN {X 0,Y 232.749,Z 430.416,A -85,B 0,C 180,E1 -22179.604,E2 -22179.604} C_VEL
LIN {X 0,Y 228.85,Z 490.415,A -85,B 0,C 180,E1 -22181.327,E2 -22181.327} C_VEL
LIN {X 0,Y 227.053,Z 504.608,A -85,B 0,C 180,E1 -22182.023,E2 -22182.023} C_VEL
LIN {X 0,Y 224.504,Z 518.083,A -85,B 0,C 180,E1 -22182.967,E2 -22182.967} C_VEL
LIN {X 0,Y 221.119,Z 531.601,A -85,B 0,C 180,E1 -22184.249,E2 -22184.249} C_VEL
LIN {X 0,Y 218.156,Z 541.791,A -85,B 0,C 180,E1 -22185.517,E2 -22185.517} C_VEL
LIN {X 0,Y 214.016,Z 553.715,A -85,B 0,C 180,E1 -22187.367,E2 -22187.367} C_VEL
LIN {X 0,Y 210.036,Z 563.601,A -85,B 0,C 180,E1 -22189.27,E2 -22189.27} C_VEL
LIN {X 0,Y 206.023,Z 572.853,A -85,B 0,C 180,E1 -22191.497,E2 -22191.497} C_VEL
LIN {X 0,Y 201.653,Z 582.09,A -85,B 0,C 180,E1 -22194.283,E2 -22194.283} C_VEL
LIN {X 0,Y 197.591,Z 589.766,A -85,B 0,C 180,E1 -22197.151,E2 -22197.151} C_VEL
LIN {X 0,Y 193.454,Z 597.138,A -85,B 0,C 180,E1 -22200.681,E2 -22200.681} C_VEL
LIN {X 0,Y 189.715,Z 603.588,A -85,B 0,C 180,E1 -22204.785,E2 -22204.785} C_VEL
LIN {X 0,Y 186.877,Z 608.454,A -85,B 0,C 180,E1 -22209.067,E2 -22209.067} C_VEL
LIN {X 0,Y 185.249,Z 611.091,A -85,B 0,C 180,E1 -22212.332,E2 -22212.332} C_VEL
LIN {X 0,Y 183.739,Z 613.373,A -85,B 0,C 180,E1 -22216.732,E2 -22216.732} C_VEL
LIN {X 0,Y 183.154,Z 614.302,A -85,B 0,C 180,E1 -22221.171,E2 -22221.171} C_VEL
LIN {X 0,Y 183.097,Z 614.271,A -85,B 0,C 180,E1 -22223.387,E2 -22223.387} C_VEL
LIN {X 0,Y 183.129,Z 613.23,A -85,B 0,C 180,E1 -22227.801,E2 -22227.801} C_VEL
LIN {X 0,Y 183.544,Z 610.869,A -85,B 0,C 180,E1 -22232.194,E2 -22232.194} C_VEL
LIN {X 0,Y 184.567,Z 607.127,A -85,B 0,C 180,E1 -22236.559,E2 -22236.559} C_VEL
LIN {X 0,Y 186.438,Z 601.86,A -85,B 0,C 180,E1 -22240.864,E2 -22240.864} C_VEL
LIN {X 0,Y 188.209,Z 596.799,A -85,B 0,C 180,E1 -22244.046,E2 -22244.046} C_VEL
LIN {X 0,Y 190.754,Z 589.572,A -85,B 0,C 180,E1 -22247.695,E2 -22247.695} C_VEL
LIN {X 0,Y 193.692,Z 581.985,A -85,B 0,C 180,E1 -22250.718,E2 -22250.718} C_VEL
LIN {X 0,Y 197.159,Z 572.878,A -85,B 0,C 180,E1 -22253.642,E2 -22253.642} C_VEL
LIN {X 0,Y 200.178,Z 563.814,A -85,B 0,C 180,E1 -22256.031,E2 -22256.031} C_VEL
LIN {X 0,Y 203.529,Z 552.999,A -85,B 0,C 180,E1 -22258.346,E2 -22258.346} C_VEL
LIN {X 0,Y 206.851,Z 541.148,A -85,B 0,C 180,E1 -22260.358,E2 -22260.358} C_VEL
LIN {X 0,Y 209.995,Z 528.024,A -85,B 0,C 180,E1 -22262.093,E2 -22262.093} C_VEL
LIN {X 0,Y 212.439,Z 515.38,A -85,B 0,C 180,E1 -22263.367,E2 -22263.367} C_VEL
LIN {X 0,Y 214.518,Z 501.072,A -85,B 0,C 180,E1 -22264.412,E2 -22264.412} C_VEL
LIN {X 0,Y 215.846,Z 487.082,A -85,B 0,C 180,E1 -22265.092,E2 -22265.092} C_VEL
LIN {X 0,Y 219.656,Z 418.592,A -85,B 0,C 180,E1 -22267.164,E2 -22267.164} C_VEL
LIN {X 0,Y 214.401,Z 406.058,A -85,B 0,C 180,E1 -22268.905,E2 -22268.905} C_VEL
LIN {X 0,Y 207.287,Z 393.342,A -85,B 0,C 180,E1 -22271.285,E2 -22271.285} C_VEL
LIN {X 0,Y 200.528,Z 382.711,A -85,B 0,C 180,E1 -22273.73,E2 -22273.73} C_VEL
LIN {X 0,Y 195.043,Z 374.842,A -85,B 0,C 180,E1 -22275.89,E2 -22275.89} C_VEL
LIN {X 0,Y 192.04,Z 370.704,A -85,B 0,C 180,E1 -22277.157,E2 -22277.157} C_VEL
LIN {X 0,Y 189.613,Z 367.53,A -85,B 0,C 180,E1 -22278.225,E2 -22278.225} C_VEL
LIN {X 0,Y 188.914,Z 366.238,A -85,B 0,C 180,E1 -22278.565,E2 -22278.565} C_VEL
LIN {X 0,Y 186.685,Z 364.201,A -85,B 0,C 180,E1 -22279.555,E2 -22279.555} C_VEL
LIN {X 0,Y 185.647,Z 361.891,A -85,B 0,C 180,E1 -22280.118,E2 -22280.118} C_VEL
LIN {X 0,Y 185.471,Z 361.006,A -85,B 0,C 180,E1 -22280.293,E2 -22280.293} C_VEL
LIN {X 0,Y 185.499,Z 361.003,A -85,B 0,C 180,E1 -22285.367,E2 -22285.367} C_VEL
LIN {X 0,Y 185.546,Z 360.995,A -85,B 0,C 180,E1 -22290.5,E2 -22290.5} C_VEL
LIN {X 0,Y 185.564,Z 360.996,A -85,B 0,C 180,E1 -22295.378,E2 -22295.378} C_VEL
LIN {X 0,Y 185.627,Z 360.952,A -85,B 0,C 180,E1 -22301.178,E2 -22301.178} C_VEL
LIN {X 0,Y 185.656,Z 360.983,A -85,B 0,C 180,E1 -22304.633,E2 -22304.633} C_VEL
LIN {X 0,Y 185.89,Z 360.907,A -85,B 0,C 180,E1 -22309.418,E2 -22309.418} C_VEL
LIN {X 0,Y 185.937,Z 360.948,A -85,B 0,C 180,E1 -22313.488,E2 -22313.488} C_VEL
LIN {X 0,Y 186.199,Z 360.913,A -85,B 0,C 180,E1 -22317.836,E2 -22317.836} C_VEL
LIN {X 0,Y 186.383,Z 360.886,A -85,B 0,C 180,E1 -22319.999,E2 -22319.999} C_VEL
LIN {X 0,Y 185.891,Z 360.951,A -85,B 0,C 180,E1 -22324.336,E2 -22324.336} C_VEL
LIN {X 0,Y 185.978,Z 360.942,A -85,B 0,C 180,E1 -22328.693,E2 -22328.693} C_VEL
LIN {X 0,Y 185.733,Z 360.971,A -85,B 0,C 180,E1 -22333.122,E2 -22333.122} C_VEL
LIN {X 0,Y 185.692,Z 360.974,A -85,B 0,C 180,E1 -22337.624,E2 -22337.624} C_VEL
LIN {X 0,Y 185.582,Z 360.987,A -85,B 0,C 180,E1 -22342.253,E2 -22342.253} C_VEL
LIN {X 0,Y 185.555,Z 360.997,A -85,B 0,C 180,E1 -22347.033,E2 -22347.033} C_VEL
LIN {X 0,Y 185.533,Z 360.998,A -85,B 0,C 180,E1 -22352.026,E2 -22352.026} C_VEL
LIN {X 0,Y 185.516,Z 361.006,A -85,B 0,C 180,E1 -22354.39,E2 -22354.39} C_VEL
LIN {X 0,Y 186.398,Z 363.648,A -85,B 0,C 180,E1 -22354.933,E2 -22354.933} C_VEL
LIN {X 0,Y 188.599,Z 365.983,A -85,B 0,C 180,E1 -22355.938,E2 -22355.938} C_VEL
LIN {X 0,Y 189.316,Z 366.709,A -85,B 0,C 180,E1 -22356.253,E2 -22356.253} C_VEL
LIN {X 0,Y 191.365,Z 369.935,A -85,B 0,C 180,E1 -22357.196,E2 -22357.196} C_VEL
LIN {X 0,Y 192.915,Z 371.799,A -85,B 0,C 180,E1 -22357.852,E2 -22357.852} C_VEL
LIN {X 0,Y 199.309,Z 382.217,A -85,B 0,C 180,E1 -22360.51,E2 -22360.51} C_VEL
LIN {X 0,Y 206.25,Z 394.935,A -85,B 0,C 180,E1 -22363.149,E2 -22363.149} C_VEL
LIN {X 0,Y 212.527,Z 408.381,A -85,B 0,C 180,E1 -22365.384,E2 -22365.384} C_VEL
LIN {X 0,Y 218.97,Z 424.67,A -85,B 0,C 180,E1 -22367.578,E2 -22367.578} C_VEL
LIN {X 0,Y 219.336,Z 427.164,A -85,B 0,C 180,E1 -22367.763,E2 -22367.763} C_VEL
LIN {X 0,Y 219.203,Z 429.512,A -85,B 0,C 180,E1 -22367.832,E2 -22367.832} C_VEL
LIN {X 0,Y 218.313,Z 435.355,A -85,B 0,C 180,E1 -22367.883,E2 -22367.883} C_VEL
LIN {X 0,Y 212.881,Z 454.367,A -85,B 0,C 180,E1 -22367.487,E2 -22367.487} C_VEL
LIN {X 0,Y 212.024,Z 460.209,A -85,B 0,C 180,E1 -22367.546,E2 -22367.546} C_VEL
LIN {X 0,Y 209.649,Z 499.447,A -85,B 0,C 180,E1 -22368.781,E2 -22368.781} C_VEL
LIN {X 0,Y 207.878,Z 514.037,A -85,B 0,C 180,E1 -22369.556,E2 -22369.556} C_VEL
LIN {X 0,Y 205.605,Z 527.441,A -85,B 0,C 180,E1 -22370.616,E2 -22370.616} C_VEL
LIN {X 0,Y 202.614,Z 540.545,A -85,B 0,C 180,E1 -22371.998,E2 -22371.998} C_VEL
LIN {X 0,Y 199.157,Z 553.234,A -85,B 0,C 180,E1 -22373.766,E2 -22373.766} C_VEL
LIN {X 0,Y 195.533,Z 565.468,A -85,B 0,C 180,E1 -22376.003,E2 -22376.003} C_VEL
LIN {X 0,Y 192.436,Z 574.445,A -85,B 0,C 180,E1 -22378.024,E2 -22378.024} C_VEL
LIN {X 0,Y 188.386,Z 585.137,A -85,B 0,C 180,E1 -22380.988,E2 -22380.988} C_VEL
LIN {X 0,Y 185.001,Z 593.967,A -85,B 0,C 180,E1 -22384.095,E2 -22384.095} C_VEL
LIN {X 0,Y 182.183,Z 601.306,A -85,B 0,C 180,E1 -22387.309,E2 -22387.309} C_VEL
LIN {X 0,Y 180.05,Z 607.421,A -85,B 0,C 180,E1 -22390.623,E2 -22390.623} C_VEL
LIN {X 0,Y 178.255,Z 612.471,A -85,B 0,C 180,E1 -22393.979,E2 -22393.979} C_VEL
LIN {X 0,Y 176.735,Z 617.672,A -85,B 0,C 180,E1 -22398.532,E2 -22398.532} C_VEL
LIN {X 0,Y 176.074,Z 621.346,A -85,B 0,C 180,E1 -22403.123,E2 -22403.123} C_VEL
